gfCNCPoint2[14445] = {X -3.6095, Y 14.8821, Z -3.0000, A 0.000, B 0.000, C 0.000 }
gfCNCPoint2[14446] = {X -3.6965, Y 14.4230, Z -3.0000, A 0.000, B 0.000, C 0.000 }
gfCNCPoint2[14447] = {X -4.2194, Y 10.4573, Z -3.0000, A 0.000, B 0.000, C 0.000 }
gfCNCPoint2[14448] = {X -7.6965, Y 10.4573, Z -3.0000, A 0.000, B 0.000, C 0.000 }
gfCNCPoint2[14449] = {X -7.6965, Y 10.4573, Z 0.0000, A 0.000, B 0.000, C 0.000 }
gfCNCPoint2[14450] = {X -7.6965, Y 10.4573, Z 11.0000, A 0.000, B 0.000, C 0.000 }
gfCNCPoint2[14451] = {X -7.9918, Y 36.0072, Z 11.0000, A 0.000, B 0.000, C 0.000 }
gfCNCPoint2[14452] = {X -7.9918, Y 36.0072, Z 0.0000, A 0.000, B 0.000, C 0.000 }
gfCNCPoint2[14453] = {X -7.9918, Y 36.0072, Z -3.0000, A 0.000, B 0.000, C 0.000 }
gfCNCPoint2[14454] = {X -4.6247, Y 35.8749, Z -3.0000, A 0.000, B 0.000, C 0.000 }
gfCNCPoint2[14455] = {X -3.6965, Y 31.9841, Z -3.0000, A 0.000, B 0.000, C 0.000 }
gfCNCPoint2[14456] = {X -3.5550, Y 31.4388, Z -3.0000, A 0.000, B 0.000, C 0.000 }
gfCNCPoint2[14457] = {X -3.3921, Y 30.8996, Z -3.0000, A 0.000, B 0.000, C 0.000 }
gfCNCPoint2[14458] = {X -3.0693, Y 30.0056, Z -3.0000, A 0.000, B 0.000, C 0.000 }
gfCNCPoint2[14459] = {X -2.6877, Y 29.1351, Z -3.0000, A 0.000, B 0.000, C 0.000 }
gfCNCPoint2[14460] = {X -1.9077, Y 27.7807, Z -3.0000, A 0.000, B 0.000, C 0.000 }
gfCNCPoint2[14461] = {X -0.9348, Y 26.5574, Z -3.0000, A 0.000, B 0.000, C 0.000 }
gfCNCPoint2[14462] = {X 0.2092, Y 25.4924, Z -3.0000, A 0.000, B 0.000, C 0.000 }
gfCNCPoint2[14463] = {X 1.4989, Y 24.6096, Z -3.0000, A 0.000, B 0.000, C 0.000 }
gfCNCPoint2[14464] = {X 1.8251, Y 24.4281, Z -3.0000, A 0.000, B 0.000, C 0.000 }
gfCNCPoint2[14465] = {X 2.1575, Y 24.2584, Z -3.0000, A 0.000, B 0.000, C 0.000 }
gfCNCPoint2[14466] = {X 1.2390, Y 23.9362, Z -3.0000, A 0.000, B 0.000, C 0.000 }
gfCNCPoint2[14467] = {X 0.4229, Y 23.4056, Z -3.0000, A 0.000, B 0.000, C 0.000 }
gfCNCPoint2[14468] = {X -0.2443, Y 22.6967, Z -3.0000, A 0.000, B 0.000, C 0.000 }
gfCNCPoint2[14469] = {X -0.7246, Y 21.8500, Z -3.0000, A 0.000, B 0.000, C 0.000 }
gfCNCPoint2[14470] = {X -3.3966, Y 15.3007, Z -3.0000, A 0.000, B 0.000, C 0.000 }
gfCNCPoint2[14471] = {X -3.6235, Y 14.3620, Z -3.0000, A 0.000, B 0.000, C 0.000 }
gfCNCPoint2[14472] = {X -3.6235, Y 13.3963, Z -3.0000, A 0.000, B 0.000, C 0.000 }
gfCNCPoint2[14473] = {X -3.3966, Y 12.4576, Z -3.0000, A 0.000, B 0.000, C 0.000 }
gfCNCPoint2[14474] = {X -2.9669, Y 11.6158, Z -3.0000, A 0.000, B 0.000, C 0.000 }
gfCNCPoint2[14475] = {X -2.3551, Y 10.8955, Z -3.0000, A 0.000, B 0.000, C 0.000 }
gfCNCPoint2[14476] = {X -1.5940, Y 10.3353, Z -3.0000, A 0.000, B 0.000, C 0.000 }
gfCNCPoint2[14477] = {X -0.9968, Y 9.9946, Z -3.0000, A 0.000, B 0.000, C 0.000 }
gfCNCPoint2[14478] = {X -0.1676, Y 9.6366, Z -3.0000, A 0.000, B 0.000, C 0.000 }
gfCNCPoint2[14479] = {X 0.7200, Y 9.4699, Z -3.0000, A 0.000, B 0.000, C 0.000 }
gfCNCPoint2[14480] = {X 1.6226, Y 9.5025, Z -3.0000, A 0.000, B 0.000, C 0.000 }
gfCNCPoint2[14481] = {X 2.4959, Y 9.7329, Z -3.0000, A 0.000, B 0.000, C 0.000 }
gfCNCPoint2[14482] = {X 2.5614, Y 9.7588, Z -3.0000, A 0.000, B 0.000, C 0.000 }
gfCNCPoint2[14483] = {X 2.6265, Y 9.7860, Z -3.0000, A 0.000, B 0.000, C 0.000 }
gfCNCPoint2[14484] = {X 3.4385, Y 9.4000, Z -3.0000, A 0.000, B 0.000, C 0.000 }
gfCNCPoint2[14485] = {X 4.2752, Y 9.0711, Z -3.0000, A 0.000, B 0.000, C 0.000 }
gfCNCPoint2[14486] = {X 6.1681, Y 8.4076, Z -3.0000, A 0.000, B 0.000, C 0.000 }
gfCNCPoint2[14487] = {X 8.1112, Y 7.9101, Z -3.0000, A 0.000, B 0.000, C 0.000 }
gfCNCPoint2[14488] = {X 10.0901, Y 7.5821, Z -3.0000, A 0.000, B 0.000, C 0.000 }
gfCNCPoint2[14489] = {X 12.0898, Y 7.4262, Z -3.0000, A 0.000, B 0.000, C 0.000 }
gfCNCPoint2[14490] = {X 14.0956, Y 7.4435, Z -3.0000, A 0.000, B 0.000, C 0.000 }
gfCNCPoint2[14491] = {X 16.0924, Y 7.6340, Z -3.0000, A 0.000, B 0.000, C 0.000 }
gfCNCPoint2[14492] = {X 17.8908, Y 7.9629, Z -3.0000, A 0.000, B 0.000, C 0.000 }
gfCNCPoint2[14493] = {X 19.6442, Y 8.4808, Z -3.0000, A 0.000, B 0.000, C 0.000 }
gfCNCPoint2[14494] = {X 21.3328, Y 9.1816, Z -3.0000, A 0.000, B 0.000, C 0.000 }
gfCNCPoint2[14495] = {X 22.9375, Y 10.0576, Z -3.0000, A 0.000, B 0.000, C 0.000 }
gfCNCPoint2[14496] = {X 24.4404, Y 11.0987, Z -3.0000, A 0.000, B 0.000, C 0.000 }
gfCNCPoint2[14497] = {X 25.5052, Y 12.0298, Z -3.0000, A 0.000, B 0.000, C 0.000 }
gfCNCPoint2[14498] = {X 26.4604, Y 13.0730, Z -3.0000, A 0.000, B 0.000, C 0.000 }
gfCNCPoint2[14499] = {X 27.2942, Y 14.2157, Z -3.0000, A 0.000, B 0.000, C 0.000 }
gfCNCPoint2[14500] = {X 27.9963, Y 15.4436, Z -3.0000, A 0.000, B 0.000, C 0.000 }
gfCNCPoint2[14501] = {X 28.5581, Y 16.7417, Z -3.0000, A 0.000, B 0.000, C 0.000 }
gfCNCPoint2[14502] = {X 29.0247, Y 18.3710, Z -3.0000, A 0.000, B 0.000, C 0.000 }
gfCNCPoint2[14503] = {X 29.3015, Y 20.0431, Z -3.0000, A 0.000, B 0.000, C 0.000 }
gfCNCPoint2[14504] = {X 29.3849, Y 21.7358, Z -3.0000, A 0.000, B 0.000, C 0.000 }
gfCNCPoint2[14505] = {X 29.2739, Y 23.4270, Z -3.0000, A 0.000, B 0.000, C 0.000 }
gfCNCPoint2[14506] = {X 28.9698, Y 25.0943, Z -3.0000, A 0.000, B 0.000, C 0.000 }
gfCNCPoint2[14507] = {X 28.5023, Y 26.6013, Z -3.0000, A 0.000, B 0.000, C 0.000 }
gfCNCPoint2[14508] = {X 27.8320, Y 28.0298, Z -3.0000, A 0.000, B 0.000, C 0.000 }
gfCNCPoint2[14509] = {X 26.9717, Y 29.3525, Z -3.0000, A 0.000, B 0.000, C 0.000 }
gfCNCPoint2[14510] = {X 25.9377, Y 30.5444, Z -3.0000, A 0.000, B 0.000, C 0.000 }
gfCNCPoint2[14511] = {X 24.7496, Y 31.5828, Z -3.0000, A 0.000, B 0.000, C 0.000 }
gfCNCPoint2[14512] = {X 25.0466, Y 31.6498, Z -3.0000, A 0.000, B 0.000, C 0.000 }
gfCNCPoint2[14513] = {X 25.3378, Y 31.7388, Z -3.0000, A 0.000, B 0.000, C 0.000 }
gfCNCPoint2[14514] = {X 26.0571, Y 32.0698, Z -3.0000, A 0.000, B 0.000, C 0.000 }
gfCNCPoint2[14515] = {X 26.6990, Y 32.5334, Z -3.0000, A 0.000, B 0.000, C 0.000 }
gfCNCPoint2[14516] = {X 27.2392, Y 33.1122, Z -3.0000, A 0.000, B 0.000, C 0.000 }
gfCNCPoint2[14517] = {X 27.6575, Y 33.7845, Z -3.0000, A 0.000, B 0.000, C 0.000 }
gfCNCPoint2[14518] = {X 30.6940, Y 40.0576, Z -3.0000, A 0.000, B 0.000, C 0.000 }
gfCNCPoint2[14519] = {X 30.9967, Y 40.9162, Z -3.0000, A 0.000, B 0.000, C 0.000 }
gfCNCPoint2[14520] = {X 31.1015, Y 41.8206, Z -3.0000, A 0.000, B 0.000, C 0.000 }
gfCNCPoint2[14521] = {X 31.0032, Y 42.7257, Z -3.0000, A 0.000, B 0.000, C 0.000 }
gfCNCPoint2[14522] = {X 30.7066, Y 43.5864, Z -3.0000, A 0.000, B 0.000, C 0.000 }
gfCNCPoint2[14523] = {X 30.2265, Y 44.3600, Z -3.0000, A 0.000, B 0.000, C 0.000 }
gfCNCPoint2[14524] = {X 29.5868, Y 45.0078, Z -3.0000, A 0.000, B 0.000, C 0.000 }
gfCNCPoint2[14525] = {X 29.0507, Y 45.4413, Z -3.0000, A 0.000, B 0.000, C 0.000 }
gfCNCPoint2[14526] = {X 28.3669, Y 45.8884, Z -3.0000, A 0.000, B 0.000, C 0.000 }
gfCNCPoint2[14527] = {X 27.6079, Y 46.1908, Z -3.0000, A 0.000, B 0.000, C 0.000 }
gfCNCPoint2[14528] = {X 26.8040, Y 46.3367, Z -3.0000, A 0.000, B 0.000, C 0.000 }
gfCNCPoint2[14529] = {X 25.9872, Y 46.3201, Z -3.0000, A 0.000, B 0.000, C 0.000 }
gfCNCPoint2[14530] = {X 25.1899, Y 46.1417, Z -3.0000, A 0.000, B 0.000, C 0.000 }
gfCNCPoint2[14531] = {X 23.5977, Y 47.0009, Z -3.0000, A 0.000, B 0.000, C 0.000 }
gfCNCPoint2[14532] = {X 21.9529, Y 47.7545, Z -3.0000, A 0.000, B 0.000, C 0.000 }
gfCNCPoint2[14533] = {X 20.2625, Y 48.3992, Z -3.0000, A 0.000, B 0.000, C 0.000 }
gfCNCPoint2[14534] = {X 18.3575, Y 49.0032, Z -3.0000, A 0.000, B 0.000, C 0.000 }
gfCNCPoint2[14535] = {X 16.4065, Y 49.4364, Z -3.0000, A 0.000, B 0.000, C 0.000 }
gfCNCPoint2[14536] = {X 14.4248, Y 49.6954, Z -3.0000, A 0.000, B 0.000, C 0.000 }
gfCNCPoint2[14537] = {X 12.4280, Y 49.7781, Z -3.0000, A 0.000, B 0.000, C 0.000 }
gfCNCPoint2[14538] = {X 10.4317, Y 49.6840, Z -3.0000, A 0.000, B 0.000, C 0.000 }
gfCNCPoint2[14539] = {X 8.4515, Y 49.4137, Z -3.0000, A 0.000, B 0.000, C 0.000 }
gfCNCPoint2[14540] = {X 6.5999, Y 48.9841, Z -3.0000, A 0.000, B 0.000, C 0.000 }
gfCNCPoint2[14541] = {X 4.8081, Y 48.3494, Z -3.0000, A 0.000, B 0.000, C 0.000 }
gfCNCPoint2[14542] = {X 3.0990, Y 47.5174, Z -3.0000, A 0.000, B 0.000, C 0.000 }
gfCNCPoint2[14543] = {X 1.4941, Y 46.4988, Z -3.0000, A 0.000, B 0.000, C 0.000 }
gfCNCPoint2[14544] = {X 0.1925, Y 45.4512, Z -3.0000, A 0.000, B 0.000, C 0.000 }
gfCNCPoint2[14545] = {X -0.9646, Y 44.2459, Z -3.0000, A 0.000, B 0.000, C 0.000 }
gfCNCPoint2[14546] = {X -1.9581, Y 42.9025, Z -3.0000, A 0.000, B 0.000, C 0.000 }
gfCNCPoint2[14547] = {X -2.7718, Y 41.4432, Z -3.0000, A 0.000, B 0.000, C 0.000 }
gfCNCPoint2[14548] = {X -3.3924, Y 39.8919, Z -3.0000, A 0.000, B 0.000, C 0.000 }
gfCNCPoint2[14549] = {X -3.5562, Y 39.3526, Z -3.0000, A 0.000, B 0.000, C 0.000 }
gfCNCPoint2[14550] = {X -3.6965, Y 38.8068, Z -3.0000, A 0.000, B 0.000, C 0.000 }
gfCNCPoint2[14551] = {X -4.6086, Y 34.9122, Z -3.0000, A 0.000, B 0.000, C 0.000 }
gfCNCPoint2[14552] = {X -7.9997, Y 34.8247, Z -3.0000, A 0.000, B 0.000, C 0.000 }
gfCNCPoint2[14553] = {X -7.9997, Y 34.8247, Z 0.0000, A 0.000, B 0.000, C 0.000 }
gfCNCPoint2[14554] = {X -7.9997, Y 34.8247, Z 11.0000, A 0.000, B 0.000, C 0.000 }
gfCNCPoint2[14555] = {X -7.9666, Y 36.4869, Z 11.0000, A 0.000, B 0.000, C 0.000 }
gfCNCPoint2[14556] = {X -7.9666, Y 36.4869, Z 0.0000, A 0.000, B 0.000, C 0.000 }
gfCNCPoint2[14557] = {X -7.9666, Y 36.4869, Z -3.0000, A 0.000, B 0.000, C 0.000 }
gfCNCPoint2[14558] = {X -4.5273, Y 36.2607, Z -3.0000, A 0.000, B 0.000, C 0.000 }
gfCNCPoint2[14559] = {X -3.6965, Y 32.3479, Z -3.0000, A 0.000, B 0.000, C 0.000 }
gfCNCPoint2[14560] = {X -3.5247, Y 31.6311, Z -3.0000, A 0.000, B 0.000, C 0.000 }
gfCNCPoint2[14561] = {X -3.3160, Y 30.9243, Z -3.0000, A 0.000, B 0.000, C 0.000 }
gfCNCPoint2[14562] = {X -2.9950, Y 30.0353, Z -3.0000, A 0.000, B 0.000, C 0.000 }
gfCNCPoint2[14563] = {X -2.6155, Y 29.1697, Z -3.0000, A 0.000, B 0.000, C 0.000 }
gfCNCPoint2[14564] = {X -1.8415, Y 27.8256, Z -3.0000, A 0.000, B 0.000, C 0.000 }
gfCNCPoint2[14565] = {X -0.8761, Y 26.6117, Z -3.0000, A 0.000, B 0.000, C 0.000 }
gfCNCPoint2[14566] = {X 0.2592, Y 25.5549, Z -3.0000, A 0.000, B 0.000, C 0.000 }
gfCNCPoint2[14567] = {X 1.5391, Y 24.6788, Z -3.0000, A 0.000, B 0.000, C 0.000 }
gfCNCPoint2[14568] = {X 1.9710, Y 24.4418, Z -3.0000, A 0.000, B 0.000, C 0.000 }
gfCNCPoint2[14569] = {X 2.4136, Y 24.2255, Z -3.0000, A 0.000, B 0.000, C 0.000 }
gfCNCPoint2[14570] = {X 1.6216, Y 24.0151, Z -3.0000, A 0.000, B 0.000, C 0.000 }
gfCNCPoint2[14571] = {X 0.8890, Y 23.6478, Z -3.0000, A 0.000, B 0.000, C 0.000 }
gfCNCPoint2[14572] = {X 0.2467, Y 23.1388, Z -3.0000, A 0.000, B 0.000, C 0.000 }
gfCNCPoint2[14573] = {X -0.2784, Y 22.5096, Z -3.0000, A 0.000, B 0.000, C 0.000 }
gfCNCPoint2[14574] = {X -0.6642, Y 21.7866, Z -3.0000, A 0.000, B 0.000, C 0.000 }
gfCNCPoint2[14575] = {X -3.2754, Y 15.3911, Z -3.0000, A 0.000, B 0.000, C 0.000 }
gfCNCPoint2[14576] = {X -3.2990, Y 15.3321, Z -3.0000, A 0.000, B 0.000, C 0.000 }
gfCNCPoint2[14577] = {X -3.3216, Y 15.2728, Z -3.0000, A 0.000, B 0.000, C 0.000 }
gfCNCPoint2[14578] = {X -3.5441, Y 14.3525, Z -3.0000, A 0.000, B 0.000, C 0.000 }
gfCNCPoint2[14579] = {X -3.5441, Y 13.4057, Z -3.0000, A 0.000, B 0.000, C 0.000 }
gfCNCPoint2[14580] = {X -3.3216, Y 12.4855, Z -3.0000, A 0.000, B 0.000, C 0.000 }
gfCNCPoint2[14581] = {X -2.9003, Y 11.6602, Z -3.0000, A 0.000, B 0.000, C 0.000 }
gfCNCPoint2[14582] = {X -2.3006, Y 10.9540, Z -3.0000, A 0.000, B 0.000, C 0.000 }
gfCNCPoint2[14583] = {X -1.5544, Y 10.4048, Z -3.0000, A 0.000, B 0.000, C 0.000 }
gfCNCPoint2[14584] = {X -0.9063, Y 10.0355, Z -3.0000, A 0.000, B 0.000, C 0.000 }
gfCNCPoint2[14585] = {X -0.1023, Y 9.7006, Z -3.0000, A 0.000, B 0.000, C 0.000 }
gfCNCPoint2[14586] = {X 0.7551, Y 9.5476, Z -3.0000, A 0.000, B 0.000, C 0.000 }
gfCNCPoint2[14587] = {X 1.6253, Y 9.5838, Z -3.0000, A 0.000, B 0.000, C 0.000 }
gfCNCPoint2[14588] = {X 2.4670, Y 9.8075, Z -3.0000, A 0.000, B 0.000, C 0.000 }
gfCNCPoint2[14589] = {X 2.5487, Y 9.8401, Z -3.0000, A 0.000, B 0.000, C 0.000 }
gfCNCPoint2[14590] = {X 2.6297, Y 9.8745, Z -3.0000, A 0.000, B 0.000, C 0.000 }
gfCNCPoint2[14591] = {X 3.4566, Y 9.4794, Z -3.0000, A 0.000, B 0.000, C 0.000 }
gfCNCPoint2[14592] = {X 4.3093, Y 9.1438, Z -3.0000, A 0.000, B 0.000, C 0.000 }
gfCNCPoint2[14593] = {X 6.1951, Y 8.4832, Z -3.0000, A 0.000, B 0.000, C 0.000 }
gfCNCPoint2[14594] = {X 8.1309, Y 7.9878, Z -3.0000, A 0.000, B 0.000, C 0.000 }
gfCNCPoint2[14595] = {X 10.1022, Y 7.6613, Z -3.0000, A 0.000, B 0.000, C 0.000 }
gfCNCPoint2[14596] = {X 12.0944, Y 7.5062, Z -3.0000, A 0.000, B 0.000, C 0.000 }
gfCNCPoint2[14597] = {X 14.0924, Y 7.5235, Z -3.0000, A 0.000, B 0.000, C 0.000 }
gfCNCPoint2[14598] = {X 16.0816, Y 7.7132, Z -3.0000, A 0.000, B 0.000, C 0.000 }
gfCNCPoint2[14599] = {X 16.4812, Y 7.7686, Z -3.0000, A 0.000, B 0.000, C 0.000 }
gfCNCPoint2[14600] = {X 18.1851, Y 8.1178, Z -3.0000, A 0.000, B 0.000, C 0.000 }
gfCNCPoint2[14601] = {X 19.8449, Y 8.6380, Z -3.0000, A 0.000, B 0.000, C 0.000 }
gfCNCPoint2[14602] = {X 21.4433, Y 9.3237, Z -3.0000, A 0.000, B 0.000, C 0.000 }
gfCNCPoint2[14603] = {X 22.9641, Y 10.1679, Z -3.0000, A 0.000, B 0.000, C 0.000 }
gfCNCPoint2[14604] = {X 24.3914, Y 11.1620, Z -3.0000, A 0.000, B 0.000, C 0.000 }
gfCNCPoint2[14605] = {X 25.4494, Y 12.0871, Z -3.0000, A 0.000, B 0.000, C 0.000 }
gfCNCPoint2[14606] = {X 26.3985, Y 13.1236, Z -3.0000, A 0.000, B 0.000, C 0.000 }
gfCNCPoint2[14607] = {X 27.2269, Y 14.2589, Z -3.0000, A 0.000, B 0.000, C 0.000 }
gfCNCPoint2[14608] = {X 27.9245, Y 15.4790, Z -3.0000, A 0.000, B 0.000, C 0.000 }
gfCNCPoint2[14609] = {X 28.4828, Y 16.7687, Z -3.0000, A 0.000, B 0.000, C 0.000 }
gfCNCPoint2[14610] = {X 28.9468, Y 18.3894, Z -3.0000, A 0.000, B 0.000, C 0.000 }
gfCNCPoint2[14611] = {X 29.2220, Y 20.0524, Z -3.0000, A 0.000, B 0.000, C 0.000 }
gfCNCPoint2[14612] = {X 29.3049, Y 21.7361, Z -3.0000, A 0.000, B 0.000, C 0.000 }
gfCNCPoint2[14613] = {X 29.1943, Y 23.4182, Z -3.0000, A 0.000, B 0.000, C 0.000 }
gfCNCPoint2[14614] = {X 28.8918, Y 25.0766, Z -3.0000, A 0.000, B 0.000, C 0.000 }
gfCNCPoint2[14615] = {X 28.4139, Y 26.6079, Z -3.0000, A 0.000, B 0.000, C 0.000 }
gfCNCPoint2[14616] = {X 27.7252, Y 28.0568, Z -3.0000, A 0.000, B 0.000, C 0.000 }
gfCNCPoint2[14617] = {X 26.8394, Y 29.3943, Z -3.0000, A 0.000, B 0.000, C 0.000 }
gfCNCPoint2[14618] = {X 25.7741, Y 30.5938, Z -3.0000, A 0.000, B 0.000, C 0.000 }
gfCNCPoint2[14619] = {X 24.5506, Y 31.6314, Z -3.0000, A 0.000, B 0.000, C 0.000 }
gfCNCPoint2[14620] = {X 24.9356, Y 31.7043, Z -3.0000, A 0.000, B 0.000, C 0.000 }
gfCNCPoint2[14621] = {X 25.3116, Y 31.8144, Z -3.0000, A 0.000, B 0.000, C 0.000 }
gfCNCPoint2[14622] = {X 26.0242, Y 32.1432, Z -3.0000, A 0.000, B 0.000, C 0.000 }
gfCNCPoint2[14623] = {X 26.6589, Y 32.6047, Z -3.0000, A 0.000, B 0.000, C 0.000 }
gfCNCPoint2[14624] = {X 27.1913, Y 33.1814, Z -3.0000, A 0.000, B 0.000, C 0.000 }
gfCNCPoint2[14625] = {X 27.6008, Y 33.8508, Z -3.0000, A 0.000, B 0.000, C 0.000 }
gfCNCPoint2[14626] = {X 30.6220, Y 40.0925, Z -3.0000, A 0.000, B 0.000, C 0.000 }
gfCNCPoint2[14627] = {X 30.9188, Y 40.9342, Z -3.0000, A 0.000, B 0.000, C 0.000 }
gfCNCPoint2[14628] = {X 31.0215, Y 41.8209, Z -3.0000, A 0.000, B 0.000, C 0.000 }
gfCNCPoint2[14629] = {X 30.9251, Y 42.7082, Z -3.0000, A 0.000, B 0.000, C 0.000 }
gfCNCPoint2[14630] = {X 30.6343, Y 43.5521, Z -3.0000, A 0.000, B 0.000, C 0.000 }
gfCNCPoint2[14631] = {X 30.1637, Y 44.3105, Z -3.0000, A 0.000, B 0.000, C 0.000 }
gfCNCPoint2[14632] = {X 29.5365, Y 44.9456, Z -3.0000, A 0.000, B 0.000, C 0.000 }
gfCNCPoint2[14633] = {X 29.0005, Y 45.3790, Z -3.0000, A 0.000, B 0.000, C 0.000 }
gfCNCPoint2[14634] = {X 28.1799, Y 45.8914, Z -3.0000, A 0.000, B 0.000, C 0.000 }
gfCNCPoint2[14635] = {X 27.2606, Y 46.1927, Z -3.0000, A 0.000, B 0.000, C 0.000 }
gfCNCPoint2[14636] = {X 26.2959, Y 46.2655, Z -3.0000, A 0.000, B 0.000, C 0.000 }
gfCNCPoint2[14637] = {X 25.3418, Y 46.1055, Z -3.0000, A 0.000, B 0.000, C 0.000 }
gfCNCPoint2[14638] = {X 25.2611, Y 46.0807, Z -3.0000, A 0.000, B 0.000, C 0.000 }
gfCNCPoint2[14639] = {X 25.1810, Y 46.0543, Z -3.0000, A 0.000, B 0.000, C 0.000 }
gfCNCPoint2[14640] = {X 23.5837, Y 46.9185, Z -3.0000, A 0.000, B 0.000, C 0.000 }
gfCNCPoint2[14641] = {X 21.9332, Y 47.6760, Z -3.0000, A 0.000, B 0.000, C 0.000 }
gfCNCPoint2[14642] = {X 20.2365, Y 48.3236, Z -3.0000, A 0.000, B 0.000, C 0.000 }
gfCNCPoint2[14643] = {X 19.5440, Y 48.5625, Z -3.0000, A 0.000, B 0.000, C 0.000 }
gfCNCPoint2[14644] = {X 17.3812, Y 49.1590, Z -3.0000, A 0.000, B 0.000, C 0.000 }
gfCNCPoint2[14645] = {X 15.1697, Y 49.5371, Z -3.0000, A 0.000, B 0.000, C 0.000 }
gfCNCPoint2[14646] = {X 12.9315, Y 49.6931, Z -3.0000, A 0.000, B 0.000, C 0.000 }
gfCNCPoint2[14647] = {X 10.6889, Y 49.6254, Z -3.0000, A 0.000, B 0.000, C 0.000 }
gfCNCPoint2[14648] = {X 8.4642, Y 49.3347, Z -3.0000, A 0.000, B 0.000, C 0.000 }
gfCNCPoint2[14649] = {X 6.6212, Y 48.9070, Z -3.0000, A 0.000, B 0.000, C 0.000 }
gfCNCPoint2[14650] = {X 4.8378, Y 48.2751, Z -3.0000, A 0.000, B 0.000, C 0.000 }
gfCNCPoint2[14651] = {X 3.1367, Y 47.4469, Z -3.0000, A 0.000, B 0.000, C 0.000 }
gfCNCPoint2[14652] = {X 1.5394, Y 46.4329, Z -3.0000, A 0.000, B 0.000, C 0.000 }
gfCNCPoint2[14653] = {X 0.2460, Y 45.3917, Z -3.0000, A 0.000, B 0.000, C 0.000 }
gfCNCPoint2[14654] = {X -0.9038, Y 44.1938, Z -3.0000, A 0.000, B 0.000, C 0.000 }
gfCNCPoint2[14655] = {X -1.8911, Y 42.8588, Z -3.0000, A 0.000, B 0.000, C 0.000 }
gfCNCPoint2[14656] = {X -2.6997, Y 41.4086, Z -3.0000, A 0.000, B 0.000, C 0.000 }
gfCNCPoint2[14657] = {X -3.3164, Y 39.8670, Z -3.0000, A 0.000, B 0.000, C 0.000 }
gfCNCPoint2[14658] = {X -3.5270, Y 39.1557, Z -3.0000, A 0.000, B 0.000, C 0.000 }
gfCNCPoint2[14659] = {X -3.6965, Y 38.4336, Z -3.0000, A 0.000, B 0.000, C 0.000 }
gfCNCPoint2[14660] = {X -4.4992, Y 34.5150, Z -3.0000, A 0.000, B 0.000, C 0.000 }
gfCNCPoint2[14661] = {X -7.9803, Y 34.3303, Z -3.0000, A 0.000, B 0.000, C 0.000 }
gfCNCPoint2[14662] = {X -7.9803, Y 34.3303, Z 0.0000, A 0.000, B 0.000, C 0.000 }
gfCNCPoint2[14663] = {X -7.9803, Y 34.3303, Z 11.0000, A 0.000, B 0.000, C 0.000 }
gfCNCPoint2[14664] = {X 39.8138, Y 26.4139, Z 11.0000, A 0.000, B 0.000, C 0.000 }
gfCNCPoint2[14665] = {X 39.8138, Y 26.4139, Z 0.0000, A 0.000, B 0.000, C 0.000 }
gfCNCPoint2[14666] = {X 39.8138, Y 26.4139, Z -3.0000, A 0.000, B 0.000, C 0.000 }
gfCNCPoint2[14667] = {X 43.6372, Y 27.8379, Z -3.0000, A 0.000, B 0.000, C 0.000 }
gfCNCPoint2[14668] = {X 48.2902, Y 15.3446, Z -3.0000, A 0.000, B 0.000, C 0.000 }
gfCNCPoint2[14669] = {X 47.9079, Y 14.6186, Z -3.0000, A 0.000, B 0.000, C 0.000 }
gfCNCPoint2[14670] = {X 47.6697, Y 13.8334, Z -3.0000, A 0.000, B 0.000, C 0.000 }
gfCNCPoint2[14671] = {X 47.5844, Y 13.0173, Z -3.0000, A 0.000, B 0.000, C 0.000 }
gfCNCPoint2[14672] = {X 47.5842, Y 12.1868, Z -3.0000, A 0.000, B 0.000, C 0.000 }
gfCNCPoint2[14673] = {X 47.6925, Y 11.2255, Z -3.0000, A 0.000, B 0.000, C 0.000 }
gfCNCPoint2[14674] = {X 48.0120, Y 10.3125, Z -3.0000, A 0.000, B 0.000, C 0.000 }
gfCNCPoint2[14675] = {X 48.5267, Y 9.4933, Z -3.0000, A 0.000, B 0.000, C 0.000 }
gfCNCPoint2[14676] = {X 49.2107, Y 8.8093, Z -3.0000, A 0.000, B 0.000, C 0.000 }
gfCNCPoint2[14677] = {X 50.0298, Y 8.2946, Z -3.0000, A 0.000, B 0.000, C 0.000 }
gfCNCPoint2[14678] = {X 50.9429, Y 7.9751, Z -3.0000, A 0.000, B 0.000, C 0.000 }
gfCNCPoint2[14679] = {X 51.9042, Y 7.8668, Z -3.0000, A 0.000, B 0.000, C 0.000 }
gfCNCPoint2[14680] = {X 59.6221, Y 7.8668, Z -3.0000, A 0.000, B 0.000, C 0.000 }
gfCNCPoint2[14681] = {X 60.5834, Y 7.9751, Z -3.0000, A 0.000, B 0.000, C 0.000 }
gfCNCPoint2[14682] = {X 61.4965, Y 8.2946, Z -3.0000, A 0.000, B 0.000, C 0.000 }
gfCNCPoint2[14683] = {X 62.3156, Y 8.8093, Z -3.0000, A 0.000, B 0.000, C 0.000 }
gfCNCPoint2[14684] = {X 62.9996, Y 9.4933, Z -3.0000, A 0.000, B 0.000, C 0.000 }
gfCNCPoint2[14685] = {X 63.5143, Y 10.3124, Z -3.0000, A 0.000, B 0.000, C 0.000 }
gfCNCPoint2[14686] = {X 63.8338, Y 11.2255, Z -3.0000, A 0.000, B 0.000, C 0.000 }
gfCNCPoint2[14687] = {X 63.9421, Y 12.1868, Z -3.0000, A 0.000, B 0.000, C 0.000 }
gfCNCPoint2[14688] = {X 63.9421, Y 12.9781, Z -3.0000, A 0.000, B 0.000, C 0.000 }
gfCNCPoint2[14689] = {X 63.8583, Y 13.8249, Z -3.0000, A 0.000, B 0.000, C 0.000 }
gfCNCPoint2[14690] = {X 63.6101, Y 14.6388, Z -3.0000, A 0.000, B 0.000, C 0.000 }
gfCNCPoint2[14691] = {X 63.2072, Y 15.3883, Z -3.0000, A 0.000, B 0.000, C 0.000 }
gfCNCPoint2[14692] = {X 63.4251, Y 15.9633, Z -3.0000, A 0.000, B 0.000, C 0.000 }
gfCNCPoint2[14693] = {X 66.0345, Y 22.8874, Z -3.0000, A 0.000, B 0.000, C 0.000 }
gfCNCPoint2[14694] = {X 72.2090, Y 39.5004, Z -3.0000, A 0.000, B 0.000, C 0.000 }
gfCNCPoint2[14695] = {X 72.5142, Y 40.2679, Z -3.0000, A 0.000, B 0.000, C 0.000 }
gfCNCPoint2[14696] = {X 73.3588, Y 40.7697, Z -3.0000, A 0.000, B 0.000, C 0.000 }
gfCNCPoint2[14697] = {X 74.0682, Y 41.4493, Z -3.0000, A 0.000, B 0.000, C 0.000 }
gfCNCPoint2[14698] = {X 74.6058, Y 42.2716, Z -3.0000, A 0.000, B 0.000, C 0.000 }
gfCNCPoint2[14699] = {X 74.9436, Y 43.1942, Z -3.0000, A 0.000, B 0.000, C 0.000 }
gfCNCPoint2[14700] = {X 75.0643, Y 44.1692, Z -3.0000, A 0.000, B 0.000, C 0.000 }
gfCNCPoint2[14701] = {X 75.0645, Y 45.0000, Z -3.0000, A 0.000, B 0.000, C 0.000 }
gfCNCPoint2[14702] = {X 74.9561, Y 45.9613, Z -3.0000, A 0.000, B 0.000, C 0.000 }
gfCNCPoint2[14703] = {X 74.6366, Y 46.8744, Z -3.0000, A 0.000, B 0.000, C 0.000 }
gfCNCPoint2[14704] = {X 74.1220, Y 47.6935, Z -3.0000, A 0.000, B 0.000, C 0.000 }
gfCNCPoint2[14705] = {X 73.4379, Y 48.3775, Z -3.0000, A 0.000, B 0.000, C 0.000 }
gfCNCPoint2[14706] = {X 72.6188, Y 48.8922, Z -3.0000, A 0.000, B 0.000, C 0.000 }
gfCNCPoint2[14707] = {X 71.7057, Y 49.2117, Z -3.0000, A 0.000, B 0.000, C 0.000 }
gfCNCPoint2[14708] = {X 70.7445, Y 49.3200, Z -3.0000, A 0.000, B 0.000, C 0.000 }
gfCNCPoint2[14709] = {X 64.1851, Y 49.3200, Z -3.0000, A 0.000, B 0.000, C 0.000 }
gfCNCPoint2[14710] = {X 63.2238, Y 49.2117, Z -3.0000, A 0.000, B 0.000, C 0.000 }
gfCNCPoint2[14711] = {X 62.3108, Y 48.8922, Z -3.0000, A 0.000, B 0.000, C 0.000 }
gfCNCPoint2[14712] = {X 61.4917, Y 48.3775, Z -3.0000, A 0.000, B 0.000, C 0.000 }
gfCNCPoint2[14713] = {X 60.8076, Y 47.6935, Z -3.0000, A 0.000, B 0.000, C 0.000 }
gfCNCPoint2[14714] = {X 60.2929, Y 46.8744, Z -3.0000, A 0.000, B 0.000, C 0.000 }
gfCNCPoint2[14715] = {X 59.9734, Y 45.9613, Z -3.0000, A 0.000, B 0.000, C 0.000 }
gfCNCPoint2[14716] = {X 59.8651, Y 45.0000, Z -3.0000, A 0.000, B 0.000, C 0.000 }
gfCNCPoint2[14717] = {X 59.8651, Y 44.2084, Z -3.0000, A 0.000, B 0.000, C 0.000 }
gfCNCPoint2[14718] = {X 59.9520, Y 43.3500, Z -3.0000, A 0.000, B 0.000, C 0.000 }
gfCNCPoint2[14719] = {X 60.2077, Y 42.5259, Z -3.0000, A 0.000, B 0.000, C 0.000 }
gfCNCPoint2[14720] = {X 60.6221, Y 41.7691, Z -3.0000, A 0.000, B 0.000, C 0.000 }
gfCNCPoint2[14721] = {X 60.0072, Y 40.0892, Z -3.0000, A 0.000, B 0.000, C 0.000 }
gfCNCPoint2[14722] = {X 52.0767, Y 40.0892, Z -3.0000, A 0.000, B 0.000, C 0.000 }
gfCNCPoint2[14723] = {X 51.3341, Y 42.0842, Z -3.0000, A 0.000, B 0.000, C 0.000 }
gfCNCPoint2[14724] = {X 51.3373, Y 42.0894, Z -3.0000, A 0.000, B 0.000, C 0.000 }
gfCNCPoint2[14725] = {X 51.6388, Y 42.7490, Z -3.0000, A 0.000, B 0.000, C 0.000 }
gfCNCPoint2[14726] = {X 51.8257, Y 43.4498, Z -3.0000, A 0.000, B 0.000, C 0.000 }
gfCNCPoint2[14727] = {X 51.8928, Y 44.1720, Z -3.0000, A 0.000, B 0.000, C 0.000 }
gfCNCPoint2[14728] = {X 51.8929, Y 45.0000, Z -3.0000, A 0.000, B 0.000, C 0.000 }
gfCNCPoint2[14729] = {X 51.7846, Y 45.9613, Z -3.0000, A 0.000, B 0.000, C 0.000 }
gfCNCPoint2[14730] = {X 51.4651, Y 46.8744, Z -3.0000, A 0.000, B 0.000, C 0.000 }
gfCNCPoint2[14731] = {X 50.9504, Y 47.6935, Z -3.0000, A 0.000, B 0.000, C 0.000 }
gfCNCPoint2[14732] = {X 50.2664, Y 48.3775, Z -3.0000, A 0.000, B 0.000, C 0.000 }
gfCNCPoint2[14733] = {X 49.4473, Y 48.8922, Z -3.0000, A 0.000, B 0.000, C 0.000 }
gfCNCPoint2[14734] = {X 48.5342, Y 49.2117, Z -3.0000, A 0.000, B 0.000, C 0.000 }
gfCNCPoint2[14735] = {X 47.5729, Y 49.3200, Z -3.0000, A 0.000, B 0.000, C 0.000 }
gfCNCPoint2[14736] = {X 40.6393, Y 49.3200, Z -3.0000, A 0.000, B 0.000, C 0.000 }
gfCNCPoint2[14737] = {X 39.6780, Y 49.2117, Z -3.0000, A 0.000, B 0.000, C 0.000 }
gfCNCPoint2[14738] = {X 38.7649, Y 48.8922, Z -3.0000, A 0.000, B 0.000, C 0.000 }
gfCNCPoint2[14739] = {X 37.9458, Y 48.3775, Z -3.0000, A 0.000, B 0.000, C 0.000 }
gfCNCPoint2[14740] = {X 37.2618, Y 47.6935, Z -3.0000, A 0.000, B 0.000, C 0.000 }
gfCNCPoint2[14741] = {X 36.7471, Y 46.8744, Z -3.0000, A 0.000, B 0.000, C 0.000 }
gfCNCPoint2[14742] = {X 36.4276, Y 45.9613, Z -3.0000, A 0.000, B 0.000, C 0.000 }
gfCNCPoint2[14743] = {X 36.3193, Y 45.0000, Z -3.0000, A 0.000, B 0.000, C 0.000 }
gfCNCPoint2[14744] = {X 36.3193, Y 44.2086, Z -3.0000, A 0.000, B 0.000, C 0.000 }
gfCNCPoint2[14745] = {X 36.4325, Y 43.2262, Z -3.0000, A 0.000, B 0.000, C 0.000 }
gfCNCPoint2[14746] = {X 36.7662, Y 42.2952, Z -3.0000, A 0.000, B 0.000, C 0.000 }
gfCNCPoint2[14747] = {X 37.3029, Y 41.4646, Z -3.0000, A 0.000, B 0.000, C 0.000 }
gfCNCPoint2[14748] = {X 38.0144, Y 40.7777, Z -3.0000, A 0.000, B 0.000, C 0.000 }
gfCNCPoint2[14749] = {X 38.8635, Y 40.2707, Z -3.0000, A 0.000, B 0.000, C 0.000 }
gfCNCPoint2[14750] = {X 38.9643, Y 40.1703, Z -3.0000, A 0.000, B 0.000, C 0.000 }
gfCNCPoint2[14751] = {X 39.5382, Y 38.8092, Z -3.0000, A 0.000, B 0.000, C 0.000 }
gfCNCPoint2[14752] = {X 40.0650, Y 37.4293, Z -3.0000, A 0.000, B 0.000, C 0.000 }
gfCNCPoint2[14753] = {X 43.6372, Y 27.8379, Z -3.0000, A 0.000, B 0.000, C 0.000 }
gfCNCPoint2[14754] = {X 39.8887, Y 26.4418, Z -3.0000, A 0.000, B 0.000, C 0.000 }
gfCNCPoint2[14755] = {X 43.7122, Y 27.8658, Z -3.0000, A 0.000, B 0.000, C 0.000 }
gfCNCPoint2[14756] = {X 48.3793, Y 15.3344, Z -3.0000, A 0.000, B 0.000, C 0.000 }
gfCNCPoint2[14757] = {X 47.9922, Y 14.6130, Z -3.0000, A 0.000, B 0.000, C 0.000 }
gfCNCPoint2[14758] = {X 47.7508, Y 13.8307, Z -3.0000, A 0.000, B 0.000, C 0.000 }
gfCNCPoint2[14759] = {X 47.6644, Y 13.0166, Z -3.0000, A 0.000, B 0.000, C 0.000 }
gfCNCPoint2[14760] = {X 47.6642, Y 12.1868, Z -3.0000, A 0.000, B 0.000, C 0.000 }
gfCNCPoint2[14761] = {X 47.7705, Y 11.2433, Z -3.0000, A 0.000, B 0.000, C 0.000 }
gfCNCPoint2[14762] = {X 48.0841, Y 10.3472, Z -3.0000, A 0.000, B 0.000, C 0.000 }
gfCNCPoint2[14763] = {X 48.5893, Y 9.5432, Z -3.0000, A 0.000, B 0.000, C 0.000 }
gfCNCPoint2[14764] = {X 49.2606, Y 8.8719, Z -3.0000, A 0.000, B 0.000, C 0.000 }
gfCNCPoint2[14765] = {X 50.0646, Y 8.3667, Z -3.0000, A 0.000, B 0.000, C 0.000 }
gfCNCPoint2[14766] = {X 50.9607, Y 8.0531, Z -3.0000, A 0.000, B 0.000, C 0.000 }
gfCNCPoint2[14767] = {X 51.9042, Y 7.9468, Z -3.0000, A 0.000, B 0.000, C 0.000 }
gfCNCPoint2[14768] = {X 59.6221, Y 7.9468, Z -3.0000, A 0.000, B 0.000, C 0.000 }
gfCNCPoint2[14769] = {X 60.5656, Y 8.0531, Z -3.0000, A 0.000, B 0.000, C 0.000 }
gfCNCPoint2[14770] = {X 61.4618, Y 8.3667, Z -3.0000, A 0.000, B 0.000, C 0.000 }
gfCNCPoint2[14771] = {X 62.2657, Y 8.8718, Z -3.0000, A 0.000, B 0.000, C 0.000 }
gfCNCPoint2[14772] = {X 62.9371, Y 9.5432, Z -3.0000, A 0.000, B 0.000, C 0.000 }
gfCNCPoint2[14773] = {X 63.4422, Y 10.3471, Z -3.0000, A 0.000, B 0.000, C 0.000 }
gfCNCPoint2[14774] = {X 63.7558, Y 11.2433, Z -3.0000, A 0.000, B 0.000, C 0.000 }
gfCNCPoint2[14775] = {X 63.8621, Y 12.1868, Z -3.0000, A 0.000, B 0.000, C 0.000 }
gfCNCPoint2[14776] = {X 63.8621, Y 12.9781, Z -3.0000, A 0.000, B 0.000, C 0.000 }
gfCNCPoint2[14777] = {X 63.7771, Y 13.8227, Z -3.0000, A 0.000, B 0.000, C 0.000 }
gfCNCPoint2[14778] = {X 63.5256, Y 14.6334, Z -3.0000, A 0.000, B 0.000, C 0.000 }
gfCNCPoint2[14779] = {X 63.1177, Y 15.3777, Z -3.0000, A 0.000, B 0.000, C 0.000 }
gfCNCPoint2[14780] = {X 63.3503, Y 15.9916, Z -3.0000, A 0.000, B 0.000, C 0.000 }
gfCNCPoint2[14781] = {X 65.9595, Y 22.9155, Z -3.0000, A 0.000, B 0.000, C 0.000 }
gfCNCPoint2[14782] = {X 72.1343, Y 39.5291, Z -3.0000, A 0.000, B 0.000, C 0.000 }
gfCNCPoint2[14783] = {X 72.4519, Y 40.3278, Z -3.0000, A 0.000, B 0.000, C 0.000 }
gfCNCPoint2[14784] = {X 73.2898, Y 40.8178, Z -3.0000, A 0.000, B 0.000, C 0.000 }
gfCNCPoint2[14785] = {X 73.9943, Y 41.4855, Z -3.0000, A 0.000, B 0.000, C 0.000 }
gfCNCPoint2[14786] = {X 74.5285, Y 42.2960, Z -3.0000, A 0.000, B 0.000, C 0.000 }
gfCNCPoint2[14787] = {X 74.8643, Y 43.2067, Z -3.0000, A 0.000, B 0.000, C 0.000 }
gfCNCPoint2[14788] = {X 74.9843, Y 44.1699, Z -3.0000, A 0.000, B 0.000, C 0.000 }
gfCNCPoint2[14789] = {X 74.9845, Y 45.0000, Z -3.0000, A 0.000, B 0.000, C 0.000 }
gfCNCPoint2[14790] = {X 74.8782, Y 45.9435, Z -3.0000, A 0.000, B 0.000, C 0.000 }
gfCNCPoint2[14791] = {X 74.5646, Y 46.8397, Z -3.0000, A 0.000, B 0.000, C 0.000 }
gfCNCPoint2[14792] = {X 74.0594, Y 47.6436, Z -3.0000, A 0.000, B 0.000, C 0.000 }
gfCNCPoint2[14793] = {X 73.3881, Y 48.3150, Z -3.0000, A 0.000, B 0.000, C 0.000 }
gfCNCPoint2[14794] = {X 72.5841, Y 48.8201, Z -3.0000, A 0.000, B 0.000, C 0.000 }
gfCNCPoint2[14795] = {X 71.6879, Y 49.1337, Z -3.0000, A 0.000, B 0.000, C 0.000 }
gfCNCPoint2[14796] = {X 70.7445, Y 49.2400, Z -3.0000, A 0.000, B 0.000, C 0.000 }
gfCNCPoint2[14797] = {X 64.1851, Y 49.2400, Z -3.0000, A 0.000, B 0.000, C 0.000 }
gfCNCPoint2[14798] = {X 63.2416, Y 49.1337, Z -3.0000, A 0.000, B 0.000, C 0.000 }
gfCNCPoint2[14799] = {X 62.3455, Y 48.8201, Z -3.0000, A 0.000, B 0.000, C 0.000 }
gfCNCPoint2[14800] = {X 61.5415, Y 48.3150, Z -3.0000, A 0.000, B 0.000, C 0.000 }
gfCNCPoint2[14801] = {X 60.8702, Y 47.6436, Z -3.0000, A 0.000, B 0.000, C 0.000 }
gfCNCPoint2[14802] = {X 60.3650, Y 46.8397, Z -3.0000, A 0.000, B 0.000, C 0.000 }
gfCNCPoint2[14803] = {X 60.0514, Y 45.9435, Z -3.0000, A 0.000, B 0.000, C 0.000 }
gfCNCPoint2[14804] = {X 59.9451, Y 45.0000, Z -3.0000, A 0.000, B 0.000, C 0.000 }
gfCNCPoint2[14805] = {X 59.9451, Y 44.2085, Z -3.0000, A 0.000, B 0.000, C 0.000 }
gfCNCPoint2[14806] = {X 60.0332, Y 43.3525, Z -3.0000, A 0.000, B 0.000, C 0.000 }
gfCNCPoint2[14807] = {X 60.2922, Y 42.5320, Z -3.0000, A 0.000, B 0.000, C 0.000 }
gfCNCPoint2[14808] = {X 60.7115, Y 41.7806, Z -3.0000, A 0.000, B 0.000, C 0.000 }
gfCNCPoint2[14809] = {X 60.0631, Y 40.0092, Z -3.0000, A 0.000, B 0.000, C 0.000 }
gfCNCPoint2[14810] = {X 52.0212, Y 40.0092, Z -3.0000, A 0.000, B 0.000, C 0.000 }
gfCNCPoint2[14811] = {X 51.2457, Y 42.0925, Z -3.0000, A 0.000, B 0.000, C 0.000 }
gfCNCPoint2[14812] = {X 51.2682, Y 42.1297, Z -3.0000, A 0.000, B 0.000, C 0.000 }
gfCNCPoint2[14813] = {X 51.5638, Y 42.7768, Z -3.0000, A 0.000, B 0.000, C 0.000 }
gfCNCPoint2[14814] = {X 51.7470, Y 43.4643, Z -3.0000, A 0.000, B 0.000, C 0.000 }
gfCNCPoint2[14815] = {X 51.8128, Y 44.1726, Z -3.0000, A 0.000, B 0.000, C 0.000 }
gfCNCPoint2[14816] = {X 51.8129, Y 45.0000, Z -3.0000, A 0.000, B 0.000, C 0.000 }
gfCNCPoint2[14817] = {X 51.7066, Y 45.9435, Z -3.0000, A 0.000, B 0.000, C 0.000 }
gfCNCPoint2[14818] = {X 51.3930, Y 46.8397, Z -3.0000, A 0.000, B 0.000, C 0.000 }
gfCNCPoint2[14819] = {X 50.8879, Y 47.6436, Z -3.0000, A 0.000, B 0.000, C 0.000 }
gfCNCPoint2[14820] = {X 50.2165, Y 48.3150, Z -3.0000, A 0.000, B 0.000, C 0.000 }
gfCNCPoint2[14821] = {X 49.4126, Y 48.8201, Z -3.0000, A 0.000, B 0.000, C 0.000 }
gfCNCPoint2[14822] = {X 48.5164, Y 49.1337, Z -3.0000, A 0.000, B 0.000, C 0.000 }
gfCNCPoint2[14823] = {X 47.5729, Y 49.2400, Z -3.0000, A 0.000, B 0.000, C 0.000 }
gfCNCPoint2[14824] = {X 40.6393, Y 49.2400, Z -3.0000, A 0.000, B 0.000, C 0.000 }
gfCNCPoint2[14825] = {X 39.6958, Y 49.1337, Z -3.0000, A 0.000, B 0.000, C 0.000 }
gfCNCPoint2[14826] = {X 38.7996, Y 48.8201, Z -3.0000, A 0.000, B 0.000, C 0.000 }
gfCNCPoint2[14827] = {X 37.9957, Y 48.3150, Z -3.0000, A 0.000, B 0.000, C 0.000 }
gfCNCPoint2[14828] = {X 37.3243, Y 47.6436, Z -3.0000, A 0.000, B 0.000, C 0.000 }
gfCNCPoint2[14829] = {X 36.8192, Y 46.8397, Z -3.0000, A 0.000, B 0.000, C 0.000 }
gfCNCPoint2[14830] = {X 36.5056, Y 45.9435, Z -3.0000, A 0.000, B 0.000, C 0.000 }
gfCNCPoint2[14831] = {X 36.3993, Y 45.0000, Z -3.0000, A 0.000, B 0.000, C 0.000 }
gfCNCPoint2[14832] = {X 36.3993, Y 44.2086, Z -3.0000, A 0.000, B 0.000, C 0.000 }
gfCNCPoint2[14833] = {X 36.5111, Y 43.2416, Z -3.0000, A 0.000, B 0.000, C 0.000 }
gfCNCPoint2[14834] = {X 36.8405, Y 42.3255, Z -3.0000, A 0.000, B 0.000, C 0.000 }
gfCNCPoint2[14835] = {X 37.3702, Y 41.5087, Z -3.0000, A 0.000, B 0.000, C 0.000 }
gfCNCPoint2[14836] = {X 38.0722, Y 40.8342, Z -3.0000, A 0.000, B 0.000, C 0.000 }
gfCNCPoint2[14837] = {X 38.9096, Y 40.3377, Z -3.0000, A 0.000, B 0.000, C 0.000 }
gfCNCPoint2[14838] = {X 39.0314, Y 40.2164, Z -3.0000, A 0.000, B 0.000, C 0.000 }
gfCNCPoint2[14839] = {X 39.6097, Y 38.8460, Z -3.0000, A 0.000, B 0.000, C 0.000 }
gfCNCPoint2[14840] = {X 40.1403, Y 37.4565, Z -3.0000, A 0.000, B 0.000, C 0.000 }
gfCNCPoint2[14841] = {X 43.7122, Y 27.8658, Z -3.0000, A 0.000, B 0.000, C 0.000 }
gfCNCPoint2[14842] = {X 39.9637, Y 26.4698, Z -3.0000, A 0.000, B 0.000, C 0.000 }
gfCNCPoint2[14843] = {X 43.7872, Y 27.8937, Z -3.0000, A 0.000, B 0.000, C 0.000 }
gfCNCPoint2[14844] = {X 48.4687, Y 15.3238, Z -3.0000, A 0.000, B 0.000, C 0.000 }
gfCNCPoint2[14845] = {X 48.0765, Y 14.6072, Z -3.0000, A 0.000, B 0.000, C 0.000 }
gfCNCPoint2[14846] = {X 47.8320, Y 13.8279, Z -3.0000, A 0.000, B 0.000, C 0.000 }
gfCNCPoint2[14847] = {X 47.7444, Y 13.0158, Z -3.0000, A 0.000, B 0.000, C 0.000 }
gfCNCPoint2[14848] = {X 47.7442, Y 12.1868, Z -3.0000, A 0.000, B 0.000, C 0.000 }
gfCNCPoint2[14849] = {X 47.8485, Y 11.2611, Z -3.0000, A 0.000, B 0.000, C 0.000 }
gfCNCPoint2[14850] = {X 48.1562, Y 10.3819, Z -3.0000, A 0.000, B 0.000, C 0.000 }
gfCNCPoint2[14851] = {X 48.6518, Y 9.5931, Z -3.0000, A 0.000, B 0.000, C 0.000 }
gfCNCPoint2[14852] = {X 49.3105, Y 8.9344, Z -3.0000, A 0.000, B 0.000, C 0.000 }
gfCNCPoint2[14853] = {X 50.0993, Y 8.4388, Z -3.0000, A 0.000, B 0.000, C 0.000 }
gfCNCPoint2[14854] = {X 50.9785, Y 8.1311, Z -3.0000, A 0.000, B 0.000, C 0.000 }
gfCNCPoint2[14855] = {X 51.9042, Y 8.0268, Z -3.0000, A 0.000, B 0.000, C 0.000 }
gfCNCPoint2[14856] = {X 59.6221, Y 8.0268, Z -3.0000, A 0.000, B 0.000, C 0.000 }
gfCNCPoint2[14857] = {X 60.5478, Y 8.1311, Z -3.0000, A 0.000, B 0.000, C 0.000 }
gfCNCPoint2[14858] = {X 61.4271, Y 8.4388, Z -3.0000, A 0.000, B 0.000, C 0.000 }
gfCNCPoint2[14859] = {X 62.2158, Y 8.9344, Z -3.0000, A 0.000, B 0.000, C 0.000 }
gfCNCPoint2[14860] = {X 62.8745, Y 9.5931, Z -3.0000, A 0.000, B 0.000, C 0.000 }
gfCNCPoint2[14861] = {X 63.3702, Y 10.3819, Z -3.0000, A 0.000, B 0.000, C 0.000 }
gfCNCPoint2[14862] = {X 63.6778, Y 11.2611, Z -3.0000, A 0.000, B 0.000, C 0.000 }
gfCNCPoint2[14863] = {X 63.7821, Y 12.1868, Z -3.0000, A 0.000, B 0.000, C 0.000 }
gfCNCPoint2[14864] = {X 63.7821, Y 12.9781, Z -3.0000, A 0.000, B 0.000, C 0.000 }
gfCNCPoint2[14865] = {X 63.6960, Y 13.8204, Z -3.0000, A 0.000, B 0.000, C 0.000 }
gfCNCPoint2[14866] = {X 63.4410, Y 14.6277, Z -3.0000, A 0.000, B 0.000, C 0.000 }
gfCNCPoint2[14867] = {X 63.0280, Y 15.3667, Z -3.0000, A 0.000, B 0.000, C 0.000 }
gfCNCPoint2[14868] = {X 63.2755, Y 16.0199, Z -3.0000, A 0.000, B 0.000, C 0.000 }
gfCNCPoint2[14869] = {X 65.8846, Y 22.9435, Z -3.0000, A 0.000, B 0.000, C 0.000 }
gfCNCPoint2[14870] = {X 72.0597, Y 39.5578, Z -3.0000, A 0.000, B 0.000, C 0.000 }
gfCNCPoint2[14871] = {X 72.3897, Y 40.3880, Z -3.0000, A 0.000, B 0.000, C 0.000 }
gfCNCPoint2[14872] = {X 73.2208, Y 40.8661, Z -3.0000, A 0.000, B 0.000, C 0.000 }
gfCNCPoint2[14873] = {X 73.9203, Y 41.5219, Z -3.0000, A 0.000, B 0.000, C 0.000 }
gfCNCPoint2[14874] = {X 74.4512, Y 42.3204, Z -3.0000, A 0.000, B 0.000, C 0.000 }
gfCNCPoint2[14875] = {X 74.7850, Y 43.2192, Z -3.0000, A 0.000, B 0.000, C 0.000 }
gfCNCPoint2[14876] = {X 74.9043, Y 44.1706, Z -3.0000, A 0.000, B 0.000, C 0.000 }
gfCNCPoint2[14877] = {X 74.9045, Y 45.0000, Z -3.0000, A 0.000, B 0.000, C 0.000 }
gfCNCPoint2[14878] = {X 74.8002, Y 45.9257, Z -3.0000, A 0.000, B 0.000, C 0.000 }
gfCNCPoint2[14879] = {X 74.4925, Y 46.8050, Z -3.0000, A 0.000, B 0.000, C 0.000 }
gfCNCPoint2[14880] = {X 73.9969, Y 47.5937, Z -3.0000, A 0.000, B 0.000, C 0.000 }
gfCNCPoint2[14881] = {X 73.3382, Y 48.2524, Z -3.0000, A 0.000, B 0.000, C 0.000 }
gfCNCPoint2[14882] = {X 72.5494, Y 48.7480, Z -3.0000, A 0.000, B 0.000, C 0.000 }
gfCNCPoint2[14883] = {X 71.6701, Y 49.0557, Z -3.0000, A 0.000, B 0.000, C 0.000 }
gfCNCPoint2[14884] = {X 70.7445, Y 49.1600, Z -3.0000, A 0.000, B 0.000, C 0.000 }
gfCNCPoint2[14885] = {X 64.1851, Y 49.1600, Z -3.0000, A 0.000, B 0.000, C 0.000 }
gfCNCPoint2[14886] = {X 63.2594, Y 49.0557, Z -3.0000, A 0.000, B 0.000, C 0.000 }
gfCNCPoint2[14887] = {X 62.3802, Y 48.7480, Z -3.0000, A 0.000, B 0.000, C 0.000 }
gfCNCPoint2[14888] = {X 61.5914, Y 48.2524, Z -3.0000, A 0.000, B 0.000, C 0.000 }
gfCNCPoint2[14889] = {X 60.9327, Y 47.5937, Z -3.0000, A 0.000, B 0.000, C 0.000 }
gfCNCPoint2[14890] = {X 60.4371, Y 46.8050, Z -3.0000, A 0.000, B 0.000, C 0.000 }
gfCNCPoint2[14891] = {X 60.1294, Y 45.9257, Z -3.0000, A 0.000, B 0.000, C 0.000 }
gfCNCPoint2[14892] = {X 60.0251, Y 45.0000, Z -3.0000, A 0.000, B 0.000, C 0.000 }
gfCNCPoint2[14893] = {X 60.0251, Y 44.2086, Z -3.0000, A 0.000, B 0.000, C 0.000 }
gfCNCPoint2[14894] = {X 60.1143, Y 43.3552, Z -3.0000, A 0.000, B 0.000, C 0.000 }
gfCNCPoint2[14895] = {X 60.3767, Y 42.5383, Z -3.0000, A 0.000, B 0.000, C 0.000 }
gfCNCPoint2[14896] = {X 60.8011, Y 41.7925, Z -3.0000, A 0.000, B 0.000, C 0.000 }
gfCNCPoint2[14897] = {X 60.1190, Y 39.9292, Z -3.0000, A 0.000, B 0.000, C 0.000 }
gfCNCPoint2[14898] = {X 51.9656, Y 39.9292, Z -3.0000, A 0.000, B 0.000, C 0.000 }
gfCNCPoint2[14899] = {X 51.1572, Y 42.1008, Z -3.0000, A 0.000, B 0.000, C 0.000 }
gfCNCPoint2[14900] = {X 51.1991, Y 42.1700, Z -3.0000, A 0.000, B 0.000, C 0.000 }
gfCNCPoint2[14901] = {X 51.4888, Y 42.8046, Z -3.0000, A 0.000, B 0.000, C 0.000 }
gfCNCPoint2[14902] = {X 51.6684, Y 43.4787, Z -3.0000, A 0.000, B 0.000, C 0.000 }
gfCNCPoint2[14903] = {X 51.7328, Y 44.1733, Z -3.0000, A 0.000, B 0.000, C 0.000 }
gfCNCPoint2[14904] = {X 51.7329, Y 45.0000, Z -3.0000, A 0.000, B 0.000, C 0.000 }
gfCNCPoint2[14905] = {X 51.6286, Y 45.9257, Z -3.0000, A 0.000, B 0.000, C 0.000 }
gfCNCPoint2[14906] = {X 51.3210, Y 46.8050, Z -3.0000, A 0.000, B 0.000, C 0.000 }
gfCNCPoint2[14907] = {X 50.8253, Y 47.5937, Z -3.0000, A 0.000, B 0.000, C 0.000 }
gfCNCPoint2[14908] = {X 50.1666, Y 48.2524, Z -3.0000, A 0.000, B 0.000, C 0.000 }
gfCNCPoint2[14909] = {X 49.3779, Y 48.7480, Z -3.0000, A 0.000, B 0.000, C 0.000 }
gfCNCPoint2[14910] = {X 48.4986, Y 49.0557, Z -3.0000, A 0.000, B 0.000, C 0.000 }
gfCNCPoint2[14911] = {X 47.5729, Y 49.1600, Z -3.0000, A 0.000, B 0.000, C 0.000 }
gfCNCPoint2[14912] = {X 40.6393, Y 49.1600, Z -3.0000, A 0.000, B 0.000, C 0.000 }
gfCNCPoint2[14913] = {X 39.7136, Y 49.0557, Z -3.0000, A 0.000, B 0.000, C 0.000 }
gfCNCPoint2[14914] = {X 38.8343, Y 48.7480, Z -3.0000, A 0.000, B 0.000, C 0.000 }
gfCNCPoint2[14915] = {X 38.0456, Y 48.2524, Z -3.0000, A 0.000, B 0.000, C 0.000 }
gfCNCPoint2[14916] = {X 37.3869, Y 47.5937, Z -3.0000, A 0.000, B 0.000, C 0.000 }
gfCNCPoint2[14917] = {X 36.8913, Y 46.8050, Z -3.0000, A 0.000, B 0.000, C 0.000 }
gfCNCPoint2[14918] = {X 36.5836, Y 45.9257, Z -3.0000, A 0.000, B 0.000, C 0.000 }
gfCNCPoint2[14919] = {X 36.4793, Y 45.0000, Z -3.0000, A 0.000, B 0.000, C 0.000 }
gfCNCPoint2[14920] = {X 36.4793, Y 44.2086, Z -3.0000, A 0.000, B 0.000, C 0.000 }
gfCNCPoint2[14921] = {X 36.5897, Y 43.2570, Z -3.0000, A 0.000, B 0.000, C 0.000 }
gfCNCPoint2[14922] = {X 36.9148, Y 42.3558, Z -3.0000, A 0.000, B 0.000, C 0.000 }
gfCNCPoint2[14923] = {X 37.4375, Y 41.5529, Z -3.0000, A 0.000, B 0.000, C 0.000 }
gfCNCPoint2[14924] = {X 38.1300, Y 40.8908, Z -3.0000, A 0.000, B 0.000, C 0.000 }
gfCNCPoint2[14925] = {X 38.9556, Y 40.4048, Z -3.0000, A 0.000, B 0.000, C 0.000 }
gfCNCPoint2[14926] = {X 39.0985, Y 40.2625, Z -3.0000, A 0.000, B 0.000, C 0.000 }
gfCNCPoint2[14927] = {X 39.6811, Y 38.8828, Z -3.0000, A 0.000, B 0.000, C 0.000 }
gfCNCPoint2[14928] = {X 40.2155, Y 37.4838, Z -3.0000, A 0.000, B 0.000, C 0.000 }
gfCNCPoint2[14929] = {X 43.7872, Y 27.8937, Z -3.0000, A 0.000, B 0.000, C 0.000 }
gfCNCPoint2[14930] = {X 40.0387, Y 26.4977, Z -3.0000, A 0.000, B 0.000, C 0.000 }
gfCNCPoint2[14931] = {X 43.8621, Y 27.9217, Z -3.0000, A 0.000, B 0.000, C 0.000 }
gfCNCPoint2[14932] = {X 48.5582, Y 15.3126, Z -3.0000, A 0.000, B 0.000, C 0.000 }
gfCNCPoint2[14933] = {X 48.1610, Y 14.6012, Z -3.0000, A 0.000, B 0.000, C 0.000 }
gfCNCPoint2[14934] = {X 47.9131, Y 13.8250, Z -3.0000, A 0.000, B 0.000, C 0.000 }
gfCNCPoint2[14935] = {X 47.8244, Y 13.0151, Z -3.0000, A 0.000, B 0.000, C 0.000 }
gfCNCPoint2[14936] = {X 47.8242, Y 12.1868, Z -3.0000, A 0.000, B 0.000, C 0.000 }
gfCNCPoint2[14937] = {X 47.9265, Y 11.2789, Z -3.0000, A 0.000, B 0.000, C 0.000 }
gfCNCPoint2[14938] = {X 48.2283, Y 10.4166, Z -3.0000, A 0.000, B 0.000, C 0.000 }
gfCNCPoint2[14939] = {X 48.7144, Y 9.6430, Z -3.0000, A 0.000, B 0.000, C 0.000 }
gfCNCPoint2[14940] = {X 49.3604, Y 8.9969, Z -3.0000, A 0.000, B 0.000, C 0.000 }
gfCNCPoint2[14941] = {X 50.1340, Y 8.5109, Z -3.0000, A 0.000, B 0.000, C 0.000 }
gfCNCPoint2[14942] = {X 50.9963, Y 8.2091, Z -3.0000, A 0.000, B 0.000, C 0.000 }
gfCNCPoint2[14943] = {X 51.9042, Y 8.1068, Z -3.0000, A 0.000, B 0.000, C 0.000 }
gfCNCPoint2[14944] = {X 59.6221, Y 8.1068, Z -3.0000, A 0.000, B 0.000, C 0.000 }
gfCNCPoint2[14945] = {X 60.5300, Y 8.2091, Z -3.0000, A 0.000, B 0.000, C 0.000 }
gfCNCPoint2[14946] = {X 61.3924, Y 8.5109, Z -3.0000, A 0.000, B 0.000, C 0.000 }
gfCNCPoint2[14947] = {X 62.1660, Y 8.9969, Z -3.0000, A 0.000, B 0.000, C 0.000 }
gfCNCPoint2[14948] = {X 62.8120, Y 9.6430, Z -3.0000, A 0.000, B 0.000, C 0.000 }
gfCNCPoint2[14949] = {X 63.2981, Y 10.4166, Z -3.0000, A 0.000, B 0.000, C 0.000 }
gfCNCPoint2[14950] = {X 63.5998, Y 11.2789, Z -3.0000, A 0.000, B 0.000, C 0.000 }
gfCNCPoint2[14951] = {X 63.7021, Y 12.1868, Z -3.0000, A 0.000, B 0.000, C 0.000 }
gfCNCPoint2[14952] = {X 63.7021, Y 12.9781, Z -3.0000, A 0.000, B 0.000, C 0.000 }
gfCNCPoint2[14953] = {X 63.6147, Y 13.8179, Z -3.0000, A 0.000, B 0.000, C 0.000 }
gfCNCPoint2[14954] = {X 63.3564, Y 14.6218, Z -3.0000, A 0.000, B 0.000, C 0.000 }
gfCNCPoint2[14955] = {X 62.9381, Y 15.3552, Z -3.0000, A 0.000, B 0.000, C 0.000 }
gfCNCPoint2[14956] = {X 63.2006, Y 16.0481, Z -3.0000, A 0.000, B 0.000, C 0.000 }
gfCNCPoint2[14957] = {X 65.8097, Y 22.9716, Z -3.0000, A 0.000, B 0.000, C 0.000 }
gfCNCPoint2[14958] = {X 71.9850, Y 39.5865, Z -3.0000, A 0.000, B 0.000, C 0.000 }
gfCNCPoint2[14959] = {X 72.3277, Y 40.4485, Z -3.0000, A 0.000, B 0.000, C 0.000 }
gfCNCPoint2[14960] = {X 73.1519, Y 40.9148, Z -3.0000, A 0.000, B 0.000, C 0.000 }
gfCNCPoint2[14961] = {X 73.8464, Y 41.5585, Z -3.0000, A 0.000, B 0.000, C 0.000 }
gfCNCPoint2[14962] = {X 74.3739, Y 42.3450, Z -3.0000, A 0.000, B 0.000, C 0.000 }
gfCNCPoint2[14963] = {X 74.7058, Y 43.2318, Z -3.0000, A 0.000, B 0.000, C 0.000 }
gfCNCPoint2[14964] = {X 74.8243, Y 44.1714, Z -3.0000, A 0.000, B 0.000, C 0.000 }
gfCNCPoint2[14965] = {X 74.8245, Y 45.0000, Z -3.0000, A 0.000, B 0.000, C 0.000 }
gfCNCPoint2[14966] = {X 74.7222, Y 45.9079, Z -3.0000, A 0.000, B 0.000, C 0.000 }
gfCNCPoint2[14967] = {X 74.4204, Y 46.7702, Z -3.0000, A 0.000, B 0.000, C 0.000 }
gfCNCPoint2[14968] = {X 73.9343, Y 47.5438, Z -3.0000, A 0.000, B 0.000, C 0.000 }
gfCNCPoint2[14969] = {X 73.2883, Y 48.1899, Z -3.0000, A 0.000, B 0.000, C 0.000 }
gfCNCPoint2[14970] = {X 72.5147, Y 48.6760, Z -3.0000, A 0.000, B 0.000, C 0.000 }
gfCNCPoint2[14971] = {X 71.6523, Y 48.9777, Z -3.0000, A 0.000, B 0.000, C 0.000 }
gfCNCPoint2[14972] = {X 70.7445, Y 49.0800, Z -3.0000, A 0.000, B 0.000, C 0.000 }
gfCNCPoint2[14973] = {X 64.1851, Y 49.0800, Z -3.0000, A 0.000, B 0.000, C 0.000 }
gfCNCPoint2[14974] = {X 63.2772, Y 48.9777, Z -3.0000, A 0.000, B 0.000, C 0.000 }
gfCNCPoint2[14975] = {X 62.4149, Y 48.6760, Z -3.0000, A 0.000, B 0.000, C 0.000 }
gfCNCPoint2[14976] = {X 61.6413, Y 48.1899, Z -3.0000, A 0.000, B 0.000, C 0.000 }
gfCNCPoint2[14977] = {X 60.9953, Y 47.5438, Z -3.0000, A 0.000, B 0.000, C 0.000 }
gfCNCPoint2[14978] = {X 60.5092, Y 46.7702, Z -3.0000, A 0.000, B 0.000, C 0.000 }
gfCNCPoint2[14979] = {X 60.2074, Y 45.9079, Z -3.0000, A 0.000, B 0.000, C 0.000 }
gfCNCPoint2[14980] = {X 60.1051, Y 45.0000, Z -3.0000, A 0.000, B 0.000, C 0.000 }
gfCNCPoint2[14981] = {X 60.1051, Y 44.2086, Z -3.0000, A 0.000, B 0.000, C 0.000 }
gfCNCPoint2[14982] = {X 60.1955, Y 43.3579, Z -3.0000, A 0.000, B 0.000, C 0.000 }
gfCNCPoint2[14983] = {X 60.4613, Y 42.5448, Z -3.0000, A 0.000, B 0.000, C 0.000 }
gfCNCPoint2[14984] = {X 60.8908, Y 41.8049, Z -3.0000, A 0.000, B 0.000, C 0.000 }
gfCNCPoint2[14985] = {X 60.1749, Y 39.8492, Z -3.0000, A 0.000, B 0.000, C 0.000 }
gfCNCPoint2[14986] = {X 51.9100, Y 39.8492, Z -3.0000, A 0.000, B 0.000, C 0.000 }
gfCNCPoint2[14987] = {X 51.0687, Y 42.1091, Z -3.0000, A 0.000, B 0.000, C 0.000 }
gfCNCPoint2[14988] = {X 51.1306, Y 42.2115, Z -3.0000, A 0.000, B 0.000, C 0.000 }
gfCNCPoint2[14989] = {X 51.4141, Y 42.8332, Z -3.0000, A 0.000, B 0.000, C 0.000 }
gfCNCPoint2[14990] = {X 51.5898, Y 43.4936, Z -3.0000, A 0.000, B 0.000, C 0.000 }
gfCNCPoint2[14991] = {X 51.6528, Y 44.1740, Z -3.0000, A 0.000, B 0.000, C 0.000 }
gfCNCPoint2[14992] = {X 51.6529, Y 45.0000, Z -3.0000, A 0.000, B 0.000, C 0.000 }
gfCNCPoint2[14993] = {X 51.5506, Y 45.9079, Z -3.0000, A 0.000, B 0.000, C 0.000 }
gfCNCPoint2[14994] = {X 51.2489, Y 46.7702, Z -3.0000, A 0.000, B 0.000, C 0.000 }
gfCNCPoint2[14995] = {X 50.7628, Y 47.5438, Z -3.0000, A 0.000, B 0.000, C 0.000 }
gfCNCPoint2[14996] = {X 50.1168, Y 48.1899, Z -3.0000, A 0.000, B 0.000, C 0.000 }
gfCNCPoint2[14997] = {X 49.3432, Y 48.6760, Z -3.0000, A 0.000, B 0.000, C 0.000 }
gfCNCPoint2[14998] = {X 48.4808, Y 48.9777, Z -3.0000, A 0.000, B 0.000, C 0.000 }
gfCNCPoint2[14999] = {X 47.5729, Y 49.0800, Z -3.0000, A 0.000, B 0.000, C 0.000 }
gfCNCPoint2[15000] = {X 40.6393, Y 49.0800, Z -3.0000, A 0.000, B 0.000, C 0.000 }
gfCNCPoint2[15001] = {X 39.7314, Y 48.9777, Z -3.0000, A 0.000, B 0.000, C 0.000 }
gfCNCPoint2[15002] = {X 38.8691, Y 48.6760, Z -3.0000, A 0.000, B 0.000, C 0.000 }
gfCNCPoint2[15003] = {X 38.0955, Y 48.1899, Z -3.0000, A 0.000, B 0.000, C 0.000 }
gfCNCPoint2[15004] = {X 37.4494, Y 47.5438, Z -3.0000, A 0.000, B 0.000, C 0.000 }
gfCNCPoint2[15005] = {X 36.9633, Y 46.7702, Z -3.0000, A 0.000, B 0.000, C 0.000 }
gfCNCPoint2[15006] = {X 36.6616, Y 45.9079, Z -3.0000, A 0.000, B 0.000, C 0.000 }
gfCNCPoint2[15007] = {X 36.5593, Y 45.0000, Z -3.0000, A 0.000, B 0.000, C 0.000 }
gfCNCPoint2[15008] = {X 36.5593, Y 44.2086, Z -3.0000, A 0.000, B 0.000, C 0.000 }
gfCNCPoint2[15009] = {X 36.6682, Y 43.2724, Z -3.0000, A 0.000, B 0.000, C 0.000 }
gfCNCPoint2[15010] = {X 36.9891, Y 42.3861, Z -3.0000, A 0.000, B 0.000, C 0.000 }
gfCNCPoint2[15011] = {X 37.5047, Y 41.5971, Z -3.0000, A 0.000, B 0.000, C 0.000 }
gfCNCPoint2[15012] = {X 38.1877, Y 40.9475, Z -3.0000, A 0.000, B 0.000, C 0.000 }
gfCNCPoint2[15013] = {X 39.0014, Y 40.4720, Z -3.0000, A 0.000, B 0.000, C 0.000 }
gfCNCPoint2[15014] = {X 39.1655, Y 40.3086, Z -3.0000, A 0.000, B 0.000, C 0.000 }
gfCNCPoint2[15015] = {X 39.7525, Y 38.9196, Z -3.0000, A 0.000, B 0.000, C 0.000 }
gfCNCPoint2[15016] = {X 40.2907, Y 37.5110, Z -3.0000, A 0.000, B 0.000, C 0.000 }
gfCNCPoint2[15017] = {X 43.8621, Y 27.9217, Z -3.0000, A 0.000, B 0.000, C 0.000 }
gfCNCPoint2[15018] = {X 40.1137, Y 26.5256, Z -3.0000, A 0.000, B 0.000, C 0.000 }
gfCNCPoint2[15019] = {X 43.9371, Y 27.9496, Z -3.0000, A 0.000, B 0.000, C 0.000 }
gfCNCPoint2[15020] = {X 48.6479, Y 15.3010, Z -3.0000, A 0.000, B 0.000, C 0.000 }
gfCNCPoint2[15021] = {X 48.2407, Y 14.5838, Z -3.0000, A 0.000, B 0.000, C 0.000 }
gfCNCPoint2[15022] = {X 47.9892, Y 13.7983, Z -3.0000, A 0.000, B 0.000, C 0.000 }
gfCNCPoint2[15023] = {X 47.9042, Y 12.9779, Z -3.0000, A 0.000, B 0.000, C 0.000 }
gfCNCPoint2[15024] = {X 47.9042, Y 12.1868, Z -3.0000, A 0.000, B 0.000, C 0.000 }
gfCNCPoint2[15025] = {X 48.0045, Y 11.2967, Z -3.0000, A 0.000, B 0.000, C 0.000 }
gfCNCPoint2[15026] = {X 48.3003, Y 10.4513, Z -3.0000, A 0.000, B 0.000, C 0.000 }
gfCNCPoint2[15027] = {X 48.7769, Y 9.6929, Z -3.0000, A 0.000, B 0.000, C 0.000 }
gfCNCPoint2[15028] = {X 49.4103, Y 9.0595, Z -3.0000, A 0.000, B 0.000, C 0.000 }
gfCNCPoint2[15029] = {X 50.1687, Y 8.5829, Z -3.0000, A 0.000, B 0.000, C 0.000 }
gfCNCPoint2[15030] = {X 51.0141, Y 8.2871, Z -3.0000, A 0.000, B 0.000, C 0.000 }
gfCNCPoint2[15031] = {X 51.9042, Y 8.1868, Z -3.0000, A 0.000, B 0.000, C 0.000 }
gfCNCPoint2[15032] = {X 59.6221, Y 8.1868, Z -3.0000, A 0.000, B 0.000, C 0.000 }
gfCNCPoint2[15033] = {X 60.5122, Y 8.2871, Z -3.0000, A 0.000, B 0.000, C 0.000 }
gfCNCPoint2[15034] = {X 61.3577, Y 8.5829, Z -3.0000, A 0.000, B 0.000, C 0.000 }
gfCNCPoint2[15035] = {X 62.1161, Y 9.0595, Z -3.0000, A 0.000, B 0.000, C 0.000 }
gfCNCPoint2[15036] = {X 62.7495, Y 9.6929, Z -3.0000, A 0.000, B 0.000, C 0.000 }
gfCNCPoint2[15037] = {X 63.2260, Y 10.4513, Z -3.0000, A 0.000, B 0.000, C 0.000 }
gfCNCPoint2[15038] = {X 63.5218, Y 11.2967, Z -3.0000, A 0.000, B 0.000, C 0.000 }
gfCNCPoint2[15039] = {X 63.6221, Y 12.1868, Z -3.0000, A 0.000, B 0.000, C 0.000 }
gfCNCPoint2[15040] = {X 63.6219, Y 13.0192, Z -3.0000, A 0.000, B 0.000, C 0.000 }
gfCNCPoint2[15041] = {X 63.5277, Y 13.8422, Z -3.0000, A 0.000, B 0.000, C 0.000 }
gfCNCPoint2[15042] = {X 63.2659, Y 14.6281, Z -3.0000, A 0.000, B 0.000, C 0.000 }
gfCNCPoint2[15043] = {X 62.8480, Y 15.3432, Z -3.0000, A 0.000, B 0.000, C 0.000 }
gfCNCPoint2[15044] = {X 63.1258, Y 16.0764, Z -3.0000, A 0.000, B 0.000, C 0.000 }
gfCNCPoint2[15045] = {X 65.7348, Y 22.9996, Z -3.0000, A 0.000, B 0.000, C 0.000 }
gfCNCPoint2[15046] = {X 71.9103, Y 39.6152, Z -3.0000, A 0.000, B 0.000, C 0.000 }
gfCNCPoint2[15047] = {X 72.2609, Y 40.4970, Z -3.0000, A 0.000, B 0.000, C 0.000 }
gfCNCPoint2[15048] = {X 72.2781, Y 40.5145, Z -3.0000, A 0.000, B 0.000, C 0.000 }
gfCNCPoint2[15049] = {X 72.3443, Y 40.5427, Z -3.0000, A 0.000, B 0.000, C 0.000 }
gfCNCPoint2[15050] = {X 72.4100, Y 40.5720, Z -3.0000, A 0.000, B 0.000, C 0.000 }
gfCNCPoint2[15051] = {X 73.1898, Y 41.0433, Z -3.0000, A 0.000, B 0.000, C 0.000 }
gfCNCPoint2[15052] = {X 73.8427, Y 41.6788, Z -3.0000, A 0.000, B 0.000, C 0.000 }
gfCNCPoint2[15053] = {X 74.3348, Y 42.4455, Z -3.0000, A 0.000, B 0.000, C 0.000 }
gfCNCPoint2[15054] = {X 74.6407, Y 43.3037, Z -3.0000, A 0.000, B 0.000, C 0.000 }
gfCNCPoint2[15055] = {X 74.7445, Y 44.2089, Z -3.0000, A 0.000, B 0.000, C 0.000 }
gfCNCPoint2[15056] = {X 74.7445, Y 45.0000, Z -3.0000, A 0.000, B 0.000, C 0.000 }
gfCNCPoint2[15057] = {X 74.6442, Y 45.8901, Z -3.0000, A 0.000, B 0.000, C 0.000 }
gfCNCPoint2[15058] = {X 74.3483, Y 46.7355, Z -3.0000, A 0.000, B 0.000, C 0.000 }
gfCNCPoint2[15059] = {X 73.8718, Y 47.4940, Z -3.0000, A 0.000, B 0.000, C 0.000 }
gfCNCPoint2[15060] = {X 73.2384, Y 48.1273, Z -3.0000, A 0.000, B 0.000, C 0.000 }
gfCNCPoint2[15061] = {X 72.4800, Y 48.6039, Z -3.0000, A 0.000, B 0.000, C 0.000 }
gfCNCPoint2[15062] = {X 71.6345, Y 48.8997, Z -3.0000, A 0.000, B 0.000, C 0.000 }
gfCNCPoint2[15063] = {X 70.7445, Y 49.0000, Z -3.0000, A 0.000, B 0.000, C 0.000 }
gfCNCPoint2[15064] = {X 64.1851, Y 49.0000, Z -3.0000, A 0.000, B 0.000, C 0.000 }
gfCNCPoint2[15065] = {X 63.2951, Y 48.8997, Z -3.0000, A 0.000, B 0.000, C 0.000 }
gfCNCPoint2[15066] = {X 62.4496, Y 48.6039, Z -3.0000, A 0.000, B 0.000, C 0.000 }
gfCNCPoint2[15067] = {X 61.6912, Y 48.1273, Z -3.0000, A 0.000, B 0.000, C 0.000 }
gfCNCPoint2[15068] = {X 61.0578, Y 47.4940, Z -3.0000, A 0.000, B 0.000, C 0.000 }
gfCNCPoint2[15069] = {X 60.5813, Y 46.7355, Z -3.0000, A 0.000, B 0.000, C 0.000 }
gfCNCPoint2[15070] = {X 60.2854, Y 45.8901, Z -3.0000, A 0.000, B 0.000, C 0.000 }
gfCNCPoint2[15071] = {X 60.1851, Y 45.0000, Z -3.0000, A 0.000, B 0.000, C 0.000 }
gfCNCPoint2[15072] = {X 60.1855, Y 44.1538, Z -3.0000, A 0.000, B 0.000, C 0.000 }
gfCNCPoint2[15073] = {X 60.2746, Y 43.3674, Z -3.0000, A 0.000, B 0.000, C 0.000 }
gfCNCPoint2[15074] = {X 60.5168, Y 42.6140, Z -3.0000, A 0.000, B 0.000, C 0.000 }
gfCNCPoint2[15075] = {X 60.9025, Y 41.9231, Z -3.0000, A 0.000, B 0.000, C 0.000 }
gfCNCPoint2[15076] = {X 60.9808, Y 41.8181, Z -3.0000, A 0.000, B 0.000, C 0.000 }
gfCNCPoint2[15077] = {X 60.2308, Y 39.7692, Z -3.0000, A 0.000, B 0.000, C 0.000 }
gfCNCPoint2[15078] = {X 51.8421, Y 39.7692, Z -3.0000, A 0.000, B 0.000, C 0.000 }
gfCNCPoint2[15079] = {X 51.8421, Y 39.8024, Z -3.0000, A 0.000, B 0.000, C 0.000 }
gfCNCPoint2[15080] = {X 50.9803, Y 42.1175, Z -3.0000, A 0.000, B 0.000, C 0.000 }
gfCNCPoint2[15081] = {X 51.0722, Y 42.2709, Z -3.0000, A 0.000, B 0.000, C 0.000 }
gfCNCPoint2[15082] = {X 51.3477, Y 42.8856, Z -3.0000, A 0.000, B 0.000, C 0.000 }
gfCNCPoint2[15083] = {X 51.5162, Y 43.5377, Z -3.0000, A 0.000, B 0.000, C 0.000 }
gfCNCPoint2[15084] = {X 51.5729, Y 44.2089, Z -3.0000, A 0.000, B 0.000, C 0.000 }
gfCNCPoint2[15085] = {X 51.5729, Y 45.0000, Z -3.0000, A 0.000, B 0.000, C 0.000 }
gfCNCPoint2[15086] = {X 51.4726, Y 45.8901, Z -3.0000, A 0.000, B 0.000, C 0.000 }
gfCNCPoint2[15087] = {X 51.1768, Y 46.7355, Z -3.0000, A 0.000, B 0.000, C 0.000 }
gfCNCPoint2[15088] = {X 50.7003, Y 47.4940, Z -3.0000, A 0.000, B 0.000, C 0.000 }
gfCNCPoint2[15089] = {X 50.0669, Y 48.1273, Z -3.0000, A 0.000, B 0.000, C 0.000 }
gfCNCPoint2[15090] = {X 49.3085, Y 48.6039, Z -3.0000, A 0.000, B 0.000, C 0.000 }
gfCNCPoint2[15091] = {X 48.4630, Y 48.8997, Z -3.0000, A 0.000, B 0.000, C 0.000 }
gfCNCPoint2[15092] = {X 47.5729, Y 49.0000, Z -3.0000, A 0.000, B 0.000, C 0.000 }
gfCNCPoint2[15093] = {X 40.6393, Y 49.0000, Z -3.0000, A 0.000, B 0.000, C 0.000 }
gfCNCPoint2[15094] = {X 39.7492, Y 48.8997, Z -3.0000, A 0.000, B 0.000, C 0.000 }
gfCNCPoint2[15095] = {X 38.9038, Y 48.6039, Z -3.0000, A 0.000, B 0.000, C 0.000 }
gfCNCPoint2[15096] = {X 38.1453, Y 48.1273, Z -3.0000, A 0.000, B 0.000, C 0.000 }
gfCNCPoint2[15097] = {X 37.5120, Y 47.4940, Z -3.0000, A 0.000, B 0.000, C 0.000 }
gfCNCPoint2[15098] = {X 37.0354, Y 46.7355, Z -3.0000, A 0.000, B 0.000, C 0.000 }
gfCNCPoint2[15099] = {X 36.7396, Y 45.8901, Z -3.0000, A 0.000, B 0.000, C 0.000 }
gfCNCPoint2[15100] = {X 36.6393, Y 45.0000, Z -3.0000, A 0.000, B 0.000, C 0.000 }
gfCNCPoint2[15101] = {X 36.6397, Y 44.1538, Z -3.0000, A 0.000, B 0.000, C 0.000 }
gfCNCPoint2[15102] = {X 36.7564, Y 43.2481, Z -3.0000, A 0.000, B 0.000, C 0.000 }
gfCNCPoint2[15103] = {X 37.0755, Y 42.3925, Z -3.0000, A 0.000, B 0.000, C 0.000 }
gfCNCPoint2[15104] = {X 37.5803, Y 41.6315, Z -3.0000, A 0.000, B 0.000, C 0.000 }
gfCNCPoint2[15105] = {X 38.2445, Y 41.0049, Z -3.0000, A 0.000, B 0.000, C 0.000 }
gfCNCPoint2[15106] = {X 39.0336, Y 40.5452, Z -3.0000, A 0.000, B 0.000, C 0.000 }
gfCNCPoint2[15107] = {X 39.0871, Y 40.5222, Z -3.0000, A 0.000, B 0.000, C 0.000 }
gfCNCPoint2[15108] = {X 39.1410, Y 40.5000, Z -3.0000, A 0.000, B 0.000, C 0.000 }
gfCNCPoint2[15109] = {X 39.1690, Y 40.4818, Z -3.0000, A 0.000, B 0.000, C 0.000 }
gfCNCPoint2[15110] = {X 39.1881, Y 40.4545, Z -3.0000, A 0.000, B 0.000, C 0.000 }
gfCNCPoint2[15111] = {X 39.2134, Y 40.3978, Z -3.0000, A 0.000, B 0.000, C 0.000 }
gfCNCPoint2[15112] = {X 39.2387, Y 40.3410, Z -3.0000, A 0.000, B 0.000, C 0.000 }
gfCNCPoint2[15113] = {X 39.8267, Y 38.9495, Z -3.0000, A 0.000, B 0.000, C 0.000 }
gfCNCPoint2[15114] = {X 40.3659, Y 37.5383, Z -3.0000, A 0.000, B 0.000, C 0.000 }
gfCNCPoint2[15115] = {X 43.9371, Y 27.9496, Z -3.0000, A 0.000, B 0.000, C 0.000 }
gfCNCPoint2[15116] = {X 40.1137, Y 26.5256, Z -3.0000, A 0.000, B 0.000, C 0.000 }
gfCNCPoint2[15117] = {X 40.1137, Y 26.5256, Z 0.0000, A 0.000, B 0.000, C 0.000 }
gfCNCPoint2[15118] = {X 40.1137, Y 26.5256, Z 11.0000, A 0.000, B 0.000, C 0.000 }
gfCNCPoint2[15119] = {X 79.0233, Y 28.5920, Z 11.0000, A 0.000, B 0.000, C 0.000 }
gfCNCPoint2[15120] = {X 79.0233, Y 28.5920, Z 0.0000, A 0.000, B 0.000, C 0.000 }
gfCNCPoint2[15121] = {X 79.0233, Y 28.5920, Z -3.0000, A 0.000, B 0.000, C 0.000 }
gfCNCPoint2[15122] = {X 83.1033, Y 28.5920, Z -3.0000, A 0.000, B 0.000, C 0.000 }
gfCNCPoint2[15123] = {X 83.1031, Y 16.2746, Z -3.0000, A 0.000, B 0.000, C 0.000 }
gfCNCPoint2[15124] = {X 82.4644, Y 15.6034, Z -3.0000, A 0.000, B 0.000, C 0.000 }
gfCNCPoint2[15125] = {X 81.9834, Y 14.8115, Z -3.0000, A 0.000, B 0.000, C 0.000 }
gfCNCPoint2[15126] = {X 81.6824, Y 13.9352, Z -3.0000, A 0.000, B 0.000, C 0.000 }
gfCNCPoint2[15127] = {X 81.5752, Y 13.0148, Z -3.0000, A 0.000, B 0.000, C 0.000 }
gfCNCPoint2[15128] = {X 81.5751, Y 12.1868, Z -3.0000, A 0.000, B 0.000, C 0.000 }
gfCNCPoint2[15129] = {X 81.6834, Y 11.2255, Z -3.0000, A 0.000, B 0.000, C 0.000 }
gfCNCPoint2[15130] = {X 82.0029, Y 10.3124, Z -3.0000, A 0.000, B 0.000, C 0.000 }
gfCNCPoint2[15131] = {X 82.5176, Y 9.4933, Z -3.0000, A 0.000, B 0.000, C 0.000 }
gfCNCPoint2[15132] = {X 83.2016, Y 8.8093, Z -3.0000, A 0.000, B 0.000, C 0.000 }
gfCNCPoint2[15133] = {X 84.0207, Y 8.2946, Z -3.0000, A 0.000, B 0.000, C 0.000 }
gfCNCPoint2[15134] = {X 84.9338, Y 7.9751, Z -3.0000, A 0.000, B 0.000, C 0.000 }
gfCNCPoint2[15135] = {X 85.8951, Y 7.8668, Z -3.0000, A 0.000, B 0.000, C 0.000 }
gfCNCPoint2[15136] = {X 94.0497, Y 7.8668, Z -3.0000, A 0.000, B 0.000, C 0.000 }
gfCNCPoint2[15137] = {X 95.0110, Y 7.9751, Z -3.0000, A 0.000, B 0.000, C 0.000 }
gfCNCPoint2[15138] = {X 95.9240, Y 8.2946, Z -3.0000, A 0.000, B 0.000, C 0.000 }
gfCNCPoint2[15139] = {X 96.7431, Y 8.8093, Z -3.0000, A 0.000, B 0.000, C 0.000 }
gfCNCPoint2[15140] = {X 97.4272, Y 9.4933, Z -3.0000, A 0.000, B 0.000, C 0.000 }
gfCNCPoint2[15141] = {X 97.9419, Y 10.3124, Z -3.0000, A 0.000, B 0.000, C 0.000 }
gfCNCPoint2[15142] = {X 98.2614, Y 11.2255, Z -3.0000, A 0.000, B 0.000, C 0.000 }
gfCNCPoint2[15143] = {X 98.3697, Y 12.1868, Z -3.0000, A 0.000, B 0.000, C 0.000 }
gfCNCPoint2[15144] = {X 98.3697, Y 12.9781, Z -3.0000, A 0.000, B 0.000, C 0.000 }
gfCNCPoint2[15145] = {X 98.2966, Y 13.7682, Z -3.0000, A 0.000, B 0.000, C 0.000 }
gfCNCPoint2[15146] = {X 98.0804, Y 14.5317, Z -3.0000, A 0.000, B 0.000, C 0.000 }
gfCNCPoint2[15147] = {X 97.7281, Y 15.2426, Z -3.0000, A 0.000, B 0.000, C 0.000 }
gfCNCPoint2[15148] = {X 101.8779, Y 25.5300, Z -3.0000, A 0.000, B 0.000, C 0.000 }
gfCNCPoint2[15149] = {X 106.0167, Y 15.2218, Z -3.0000, A 0.000, B 0.000, C 0.000 }
gfCNCPoint2[15150] = {X 105.6762, Y 14.5288, Z -3.0000, A 0.000, B 0.000, C 0.000 }
gfCNCPoint2[15151] = {X 105.4646, Y 13.7863, Z -3.0000, A 0.000, B 0.000, C 0.000 }
gfCNCPoint2[15152] = {X 105.3885, Y 13.0179, Z -3.0000, A 0.000, B 0.000, C 0.000 }
gfCNCPoint2[15153] = {X 105.3883, Y 12.1868, Z -3.0000, A 0.000, B 0.000, C 0.000 }
gfCNCPoint2[15154] = {X 105.4966, Y 11.2255, Z -3.0000, A 0.000, B 0.000, C 0.000 }
gfCNCPoint2[15155] = {X 105.8161, Y 10.3124, Z -3.0000, A 0.000, B 0.000, C 0.000 }
gfCNCPoint2[15156] = {X 106.3308, Y 9.4933, Z -3.0000, A 0.000, B 0.000, C 0.000 }
gfCNCPoint2[15157] = {X 107.0148, Y 8.8093, Z -3.0000, A 0.000, B 0.000, C 0.000 }
gfCNCPoint2[15158] = {X 107.8339, Y 8.2946, Z -3.0000, A 0.000, B 0.000, C 0.000 }
gfCNCPoint2[15159] = {X 108.7470, Y 7.9751, Z -3.0000, A 0.000, B 0.000, C 0.000 }
gfCNCPoint2[15160] = {X 109.7083, Y 7.8668, Z -3.0000, A 0.000, B 0.000, C 0.000 }
gfCNCPoint2[15161] = {X 117.7916, Y 7.8668, Z -3.0000, A 0.000, B 0.000, C 0.000 }
gfCNCPoint2[15162] = {X 118.7529, Y 7.9751, Z -3.0000, A 0.000, B 0.000, C 0.000 }
gfCNCPoint2[15163] = {X 119.6660, Y 8.2946, Z -3.0000, A 0.000, B 0.000, C 0.000 }
gfCNCPoint2[15164] = {X 120.4851, Y 8.8093, Z -3.0000, A 0.000, B 0.000, C 0.000 }
gfCNCPoint2[15165] = {X 121.1691, Y 9.4933, Z -3.0000, A 0.000, B 0.000, C 0.000 }
gfCNCPoint2[15166] = {X 121.6838, Y 10.3124, Z -3.0000, A 0.000, B 0.000, C 0.000 }
gfCNCPoint2[15167] = {X 122.0033, Y 11.2255, Z -3.0000, A 0.000, B 0.000, C 0.000 }
gfCNCPoint2[15168] = {X 122.1116, Y 12.1868, Z -3.0000, A 0.000, B 0.000, C 0.000 }
gfCNCPoint2[15169] = {X 122.1116, Y 12.9781, Z -3.0000, A 0.000, B 0.000, C 0.000 }
gfCNCPoint2[15170] = {X 122.0103, Y 13.9079, Z -3.0000, A 0.000, B 0.000, C 0.000 }
gfCNCPoint2[15171] = {X 121.7113, Y 14.7941, Z -3.0000, A 0.000, B 0.000, C 0.000 }
gfCNCPoint2[15172] = {X 121.2285, Y 15.5952, Z -3.0000, A 0.000, B 0.000, C 0.000 }
gfCNCPoint2[15173] = {X 120.5847, Y 16.2736, Z -3.0000, A 0.000, B 0.000, C 0.000 }
gfCNCPoint2[15174] = {X 120.5834, Y 40.9139, Z -3.0000, A 0.000, B 0.000, C 0.000 }
gfCNCPoint2[15175] = {X 120.6219, Y 40.9451, Z -3.0000, A 0.000, B 0.000, C 0.000 }
gfCNCPoint2[15176] = {X 121.2454, Y 41.6139, Z -3.0000, A 0.000, B 0.000, C 0.000 }
gfCNCPoint2[15177] = {X 121.7142, Y 42.3989, Z -3.0000, A 0.000, B 0.000, C 0.000 }
gfCNCPoint2[15178] = {X 122.0072, Y 43.2650, Z -3.0000, A 0.000, B 0.000, C 0.000 }
gfCNCPoint2[15179] = {X 122.1114, Y 44.1734, Z -3.0000, A 0.000, B 0.000, C 0.000 }
gfCNCPoint2[15180] = {X 122.1116, Y 45.0000, Z -3.0000, A 0.000, B 0.000, C 0.000 }
gfCNCPoint2[15181] = {X 122.0033, Y 45.9613, Z -3.0000, A 0.000, B 0.000, C 0.000 }
gfCNCPoint2[15182] = {X 121.6838, Y 46.8744, Z -3.0000, A 0.000, B 0.000, C 0.000 }
gfCNCPoint2[15183] = {X 121.1691, Y 47.6935, Z -3.0000, A 0.000, B 0.000, C 0.000 }
gfCNCPoint2[15184] = {X 120.4851, Y 48.3775, Z -3.0000, A 0.000, B 0.000, C 0.000 }
gfCNCPoint2[15185] = {X 119.6660, Y 48.8922, Z -3.0000, A 0.000, B 0.000, C 0.000 }
gfCNCPoint2[15186] = {X 118.7529, Y 49.2117, Z -3.0000, A 0.000, B 0.000, C 0.000 }
gfCNCPoint2[15187] = {X 117.7916, Y 49.3200, Z -3.0000, A 0.000, B 0.000, C 0.000 }
gfCNCPoint2[15188] = {X 111.9185, Y 49.3200, Z -3.0000, A 0.000, B 0.000, C 0.000 }
gfCNCPoint2[15189] = {X 110.9619, Y 49.2128, Z -3.0000, A 0.000, B 0.000, C 0.000 }
gfCNCPoint2[15190] = {X 110.0529, Y 48.8964, Z -3.0000, A 0.000, B 0.000, C 0.000 }
gfCNCPoint2[15191] = {X 109.2365, Y 48.3866, Z -3.0000, A 0.000, B 0.000, C 0.000 }
gfCNCPoint2[15192] = {X 108.5532, Y 47.7087, Z -3.0000, A 0.000, B 0.000, C 0.000 }
gfCNCPoint2[15193] = {X 108.0369, Y 46.8963, Z -3.0000, A 0.000, B 0.000, C 0.000 }
gfCNCPoint2[15194] = {X 107.7134, Y 45.9898, Z -3.0000, A 0.000, B 0.000, C 0.000 }
gfCNCPoint2[15195] = {X 107.5986, Y 45.0341, Z -3.0000, A 0.000, B 0.000, C 0.000 }
gfCNCPoint2[15196] = {X 107.5985, Y 44.1811, Z -3.0000, A 0.000, B 0.000, C 0.000 }
gfCNCPoint2[15197] = {X 107.6344, Y 43.6356, Z -3.0000, A 0.000, B 0.000, C 0.000 }
gfCNCPoint2[15198] = {X 107.7417, Y 43.0994, Z -3.0000, A 0.000, B 0.000, C 0.000 }
gfCNCPoint2[15199] = {X 107.9081, Y 42.6068, Z -3.0000, A 0.000, B 0.000, C 0.000 }
gfCNCPoint2[15200] = {X 108.1348, Y 42.1387, Z -3.0000, A 0.000, B 0.000, C 0.000 }
gfCNCPoint2[15201] = {X 108.5861, Y 41.4658, Z -3.0000, A 0.000, B 0.000, C 0.000 }
gfCNCPoint2[15202] = {X 109.1266, Y 40.8623, Z -3.0000, A 0.000, B 0.000, C 0.000 }
gfCNCPoint2[15203] = {X 109.1265, Y 39.2945, Z -3.0000, A 0.000, B 0.000, C 0.000 }
gfCNCPoint2[15204] = {X 106.1118, Y 46.6615, Z -3.0000, A 0.000, B 0.000, C 0.000 }
gfCNCPoint2[15205] = {X 105.7417, Y 47.3611, Z -3.0000, A 0.000, B 0.000, C 0.000 }
gfCNCPoint2[15206] = {X 105.2502, Y 47.9815, Z -3.0000, A 0.000, B 0.000, C 0.000 }
gfCNCPoint2[15207] = {X 104.6538, Y 48.5018, Z -3.0000, A 0.000, B 0.000, C 0.000 }
gfCNCPoint2[15208] = {X 103.9724, Y 48.9046, Z -3.0000, A 0.000, B 0.000, C 0.000 }
gfCNCPoint2[15209] = {X 103.0287, Y 49.2242, Z -3.0000, A 0.000, B 0.000, C 0.000 }
gfCNCPoint2[15210] = {X 102.0368, Y 49.3191, Z -3.0000, A 0.000, B 0.000, C 0.000 }
gfCNCPoint2[15211] = {X 101.0496, Y 49.1842, Z -3.0000, A 0.000, B 0.000, C 0.000 }
gfCNCPoint2[15212] = {X 100.1195, Y 48.8268, Z -3.0000, A 0.000, B 0.000, C 0.000 }
gfCNCPoint2[15213] = {X 99.2961, Y 48.2657, Z -3.0000, A 0.000, B 0.000, C 0.000 }
gfCNCPoint2[15214] = {X 98.6231, Y 47.5309, Z -3.0000, A 0.000, B 0.000, C 0.000 }
gfCNCPoint2[15215] = {X 98.1363, Y 46.6615, Z -3.0000, A 0.000, B 0.000, C 0.000 }
gfCNCPoint2[15216] = {X 95.1304, Y 39.3101, Z -3.0000, A 0.000, B 0.000, C 0.000 }
gfCNCPoint2[15217] = {X 95.1305, Y 40.9053, Z -3.0000, A 0.000, B 0.000, C 0.000 }
gfCNCPoint2[15218] = {X 95.6595, Y 41.4476, Z -3.0000, A 0.000, B 0.000, C 0.000 }
gfCNCPoint2[15219] = {X 96.0877, Y 42.0725, Z -3.0000, A 0.000, B 0.000, C 0.000 }
gfCNCPoint2[15220] = {X 96.3309, Y 42.5741, Z -3.0000, A 0.000, B 0.000, C 0.000 }
gfCNCPoint2[15221] = {X 96.5088, Y 43.1024, Z -3.0000, A 0.000, B 0.000, C 0.000 }
gfCNCPoint2[15222] = {X 96.6187, Y 43.6496, Z -3.0000, A 0.000, B 0.000, C 0.000 }
gfCNCPoint2[15223] = {X 96.6585, Y 44.2063, Z -3.0000, A 0.000, B 0.000, C 0.000 }
gfCNCPoint2[15224] = {X 96.6583, Y 45.0415, Z -3.0000, A 0.000, B 0.000, C 0.000 }
gfCNCPoint2[15225] = {X 96.5422, Y 45.9960, Z -3.0000, A 0.000, B 0.000, C 0.000 }
gfCNCPoint2[15226] = {X 96.2178, Y 46.9011, Z -3.0000, A 0.000, B 0.000, C 0.000 }
gfCNCPoint2[15227] = {X 95.7012, Y 47.7120, Z -3.0000, A 0.000, B 0.000, C 0.000 }
gfCNCPoint2[15228] = {X 95.0181, Y 48.3886, Z -3.0000, A 0.000, B 0.000, C 0.000 }
gfCNCPoint2[15229] = {X 94.2022, Y 48.8973, Z -3.0000, A 0.000, B 0.000, C 0.000 }
gfCNCPoint2[15230] = {X 93.2940, Y 49.2130, Z -3.0000, A 0.000, B 0.000, C 0.000 }
gfCNCPoint2[15231] = {X 92.3385, Y 49.3200, Z -3.0000, A 0.000, B 0.000, C 0.000 }
gfCNCPoint2[15232] = {X 85.8951, Y 49.3200, Z -3.0000, A 0.000, B 0.000, C 0.000 }
gfCNCPoint2[15233] = {X 84.9387, Y 49.2128, Z -3.0000, A 0.000, B 0.000, C 0.000 }
gfCNCPoint2[15234] = {X 84.0297, Y 48.8965, Z -3.0000, A 0.000, B 0.000, C 0.000 }
gfCNCPoint2[15235] = {X 83.2134, Y 48.3869, Z -3.0000, A 0.000, B 0.000, C 0.000 }
gfCNCPoint2[15236] = {X 82.5301, Y 47.7091, Z -3.0000, A 0.000, B 0.000, C 0.000 }
gfCNCPoint2[15237] = {X 82.0138, Y 46.8970, Z -3.0000, A 0.000, B 0.000, C 0.000 }
gfCNCPoint2[15238] = {X 81.6902, Y 45.9906, Z -3.0000, A 0.000, B 0.000, C 0.000 }
gfCNCPoint2[15239] = {X 81.5752, Y 45.0351, Z -3.0000, A 0.000, B 0.000, C 0.000 }
gfCNCPoint2[15240] = {X 81.5751, Y 44.2069, Z -3.0000, A 0.000, B 0.000, C 0.000 }
gfCNCPoint2[15241] = {X 81.6807, Y 43.2777, Z -3.0000, A 0.000, B 0.000, C 0.000 }
gfCNCPoint2[15242] = {X 81.9812, Y 42.3922, Z -3.0000, A 0.000, B 0.000, C 0.000 }
gfCNCPoint2[15243] = {X 82.4627, Y 41.5905, Z -3.0000, A 0.000, B 0.000, C 0.000 }
gfCNCPoint2[15244] = {X 83.1034, Y 40.9093, Z -3.0000, A 0.000, B 0.000, C 0.000 }
gfCNCPoint2[15245] = {X 83.1033, Y 28.5920, Z -3.0000, A 0.000, B 0.000, C 0.000 }
gfCNCPoint2[15246] = {X 79.1033, Y 28.5920, Z -3.0000, A 0.000, B 0.000, C 0.000 }
gfCNCPoint2[15247] = {X 83.1833, Y 28.5920, Z -3.0000, A 0.000, B 0.000, C 0.000 }
gfCNCPoint2[15248] = {X 83.1831, Y 16.2373, Z -3.0000, A 0.000, B 0.000, C 0.000 }
gfCNCPoint2[15249] = {X 82.5448, Y 15.5767, Z -3.0000, A 0.000, B 0.000, C 0.000 }
gfCNCPoint2[15250] = {X 82.0637, Y 14.7942, Z -3.0000, A 0.000, B 0.000, C 0.000 }
gfCNCPoint2[15251] = {X 81.7625, Y 13.9264, Z -3.0000, A 0.000, B 0.000, C 0.000 }
gfCNCPoint2[15252] = {X 81.6552, Y 13.0142, Z -3.0000, A 0.000, B 0.000, C 0.000 }
gfCNCPoint2[15253] = {X 81.6551, Y 12.1868, Z -3.0000, A 0.000, B 0.000, C 0.000 }
gfCNCPoint2[15254] = {X 81.7614, Y 11.2433, Z -3.0000, A 0.000, B 0.000, C 0.000 }
gfCNCPoint2[15255] = {X 82.0750, Y 10.3472, Z -3.0000, A 0.000, B 0.000, C 0.000 }
gfCNCPoint2[15256] = {X 82.5801, Y 9.5432, Z -3.0000, A 0.000, B 0.000, C 0.000 }
gfCNCPoint2[15257] = {X 83.2515, Y 8.8719, Z -3.0000, A 0.000, B 0.000, C 0.000 }
gfCNCPoint2[15258] = {X 84.0554, Y 8.3667, Z -3.0000, A 0.000, B 0.000, C 0.000 }
gfCNCPoint2[15259] = {X 84.9516, Y 8.0531, Z -3.0000, A 0.000, B 0.000, C 0.000 }
gfCNCPoint2[15260] = {X 85.8951, Y 7.9468, Z -3.0000, A 0.000, B 0.000, C 0.000 }
gfCNCPoint2[15261] = {X 94.0497, Y 7.9468, Z -3.0000, A 0.000, B 0.000, C 0.000 }
gfCNCPoint2[15262] = {X 94.9932, Y 8.0531, Z -3.0000, A 0.000, B 0.000, C 0.000 }
gfCNCPoint2[15263] = {X 95.8893, Y 8.3667, Z -3.0000, A 0.000, B 0.000, C 0.000 }
gfCNCPoint2[15264] = {X 96.6933, Y 8.8718, Z -3.0000, A 0.000, B 0.000, C 0.000 }
gfCNCPoint2[15265] = {X 97.3646, Y 9.5432, Z -3.0000, A 0.000, B 0.000, C 0.000 }
gfCNCPoint2[15266] = {X 97.8698, Y 10.3471, Z -3.0000, A 0.000, B 0.000, C 0.000 }
gfCNCPoint2[15267] = {X 98.1834, Y 11.2433, Z -3.0000, A 0.000, B 0.000, C 0.000 }
gfCNCPoint2[15268] = {X 98.2897, Y 12.1868, Z -3.0000, A 0.000, B 0.000, C 0.000 }
gfCNCPoint2[15269] = {X 98.2897, Y 12.9781, Z -3.0000, A 0.000, B 0.000, C 0.000 }
gfCNCPoint2[15270] = {X 98.2155, Y 13.7668, Z -3.0000, A 0.000, B 0.000, C 0.000 }
gfCNCPoint2[15271] = {X 97.9960, Y 14.5279, Z -3.0000, A 0.000, B 0.000, C 0.000 }
gfCNCPoint2[15272] = {X 97.6387, Y 15.2348, Z -3.0000, A 0.000, B 0.000, C 0.000 }
gfCNCPoint2[15273] = {X 101.8779, Y 25.7436, Z -3.0000, A 0.000, B 0.000, C 0.000 }
gfCNCPoint2[15274] = {X 101.9522, Y 25.5598, Z -3.0000, A 0.000, B 0.000, C 0.000 }
gfCNCPoint2[15275] = {X 106.1059, Y 15.2143, Z -3.0000, A 0.000, B 0.000, C 0.000 }
gfCNCPoint2[15276] = {X 105.7605, Y 14.5249, Z -3.0000, A 0.000, B 0.000, C 0.000 }
gfCNCPoint2[15277] = {X 105.5457, Y 13.7844, Z -3.0000, A 0.000, B 0.000, C 0.000 }
gfCNCPoint2[15278] = {X 105.4685, Y 13.0172, Z -3.0000, A 0.000, B 0.000, C 0.000 }
gfCNCPoint2[15279] = {X 105.4683, Y 12.1868, Z -3.0000, A 0.000, B 0.000, C 0.000 }
gfCNCPoint2[15280] = {X 105.5746, Y 11.2433, Z -3.0000, A 0.000, B 0.000, C 0.000 }
gfCNCPoint2[15281] = {X 105.8882, Y 10.3471, Z -3.0000, A 0.000, B 0.000, C 0.000 }
gfCNCPoint2[15282] = {X 106.3933, Y 9.5432, Z -3.0000, A 0.000, B 0.000, C 0.000 }
gfCNCPoint2[15283] = {X 107.0647, Y 8.8718, Z -3.0000, A 0.000, B 0.000, C 0.000 }
gfCNCPoint2[15284] = {X 107.8686, Y 8.3667, Z -3.0000, A 0.000, B 0.000, C 0.000 }
gfCNCPoint2[15285] = {X 108.7648, Y 8.0531, Z -3.0000, A 0.000, B 0.000, C 0.000 }
gfCNCPoint2[15286] = {X 109.7083, Y 7.9468, Z -3.0000, A 0.000, B 0.000, C 0.000 }
gfCNCPoint2[15287] = {X 117.7916, Y 7.9468, Z -3.0000, A 0.000, B 0.000, C 0.000 }
gfCNCPoint2[15288] = {X 118.7351, Y 8.0531, Z -3.0000, A 0.000, B 0.000, C 0.000 }
gfCNCPoint2[15289] = {X 119.6312, Y 8.3667, Z -3.0000, A 0.000, B 0.000, C 0.000 }
gfCNCPoint2[15290] = {X 120.4352, Y 8.8718, Z -3.0000, A 0.000, B 0.000, C 0.000 }
gfCNCPoint2[15291] = {X 121.1065, Y 9.5432, Z -3.0000, A 0.000, B 0.000, C 0.000 }
gfCNCPoint2[15292] = {X 121.6117, Y 10.3471, Z -3.0000, A 0.000, B 0.000, C 0.000 }
gfCNCPoint2[15293] = {X 121.9253, Y 11.2433, Z -3.0000, A 0.000, B 0.000, C 0.000 }
gfCNCPoint2[15294] = {X 122.0316, Y 12.1868, Z -3.0000, A 0.000, B 0.000, C 0.000 }
gfCNCPoint2[15295] = {X 122.0316, Y 12.9781, Z -3.0000, A 0.000, B 0.000, C 0.000 }
gfCNCPoint2[15296] = {X 121.9302, Y 13.8997, Z -3.0000, A 0.000, B 0.000, C 0.000 }
gfCNCPoint2[15297] = {X 121.6309, Y 14.7772, Z -3.0000, A 0.000, B 0.000, C 0.000 }
gfCNCPoint2[15298] = {X 121.1480, Y 15.5687, Z -3.0000, A 0.000, B 0.000, C 0.000 }
gfCNCPoint2[15299] = {X 120.5047, Y 16.2363, Z -3.0000, A 0.000, B 0.000, C 0.000 }
gfCNCPoint2[15300] = {X 120.5034, Y 40.9519, Z -3.0000, A 0.000, B 0.000, C 0.000 }
gfCNCPoint2[15301] = {X 120.5704, Y 41.0063, Z -3.0000, A 0.000, B 0.000, C 0.000 }
gfCNCPoint2[15302] = {X 121.1820, Y 41.6627, Z -3.0000, A 0.000, B 0.000, C 0.000 }
gfCNCPoint2[15303] = {X 121.6418, Y 42.4330, Z -3.0000, A 0.000, B 0.000, C 0.000 }
gfCNCPoint2[15304] = {X 121.9292, Y 43.2828, Z -3.0000, A 0.000, B 0.000, C 0.000 }
gfCNCPoint2[15305] = {X 122.0314, Y 44.1740, Z -3.0000, A 0.000, B 0.000, C 0.000 }
gfCNCPoint2[15306] = {X 122.0316, Y 45.0000, Z -3.0000, A 0.000, B 0.000, C 0.000 }
gfCNCPoint2[15307] = {X 121.9253, Y 45.9435, Z -3.0000, A 0.000, B 0.000, C 0.000 }
gfCNCPoint2[15308] = {X 121.6117, Y 46.8397, Z -3.0000, A 0.000, B 0.000, C 0.000 }
gfCNCPoint2[15309] = {X 121.1065, Y 47.6436, Z -3.0000, A 0.000, B 0.000, C 0.000 }
gfCNCPoint2[15310] = {X 120.4352, Y 48.3150, Z -3.0000, A 0.000, B 0.000, C 0.000 }
gfCNCPoint2[15311] = {X 119.6312, Y 48.8201, Z -3.0000, A 0.000, B 0.000, C 0.000 }
gfCNCPoint2[15312] = {X 118.7351, Y 49.1337, Z -3.0000, A 0.000, B 0.000, C 0.000 }
gfCNCPoint2[15313] = {X 117.7916, Y 49.2400, Z -3.0000, A 0.000, B 0.000, C 0.000 }
gfCNCPoint2[15314] = {X 111.9185, Y 49.2400, Z -3.0000, A 0.000, B 0.000, C 0.000 }
gfCNCPoint2[15315] = {X 110.9797, Y 49.1348, Z -3.0000, A 0.000, B 0.000, C 0.000 }
gfCNCPoint2[15316] = {X 110.0874, Y 48.8242, Z -3.0000, A 0.000, B 0.000, C 0.000 }
gfCNCPoint2[15317] = {X 109.2861, Y 48.3239, Z -3.0000, A 0.000, B 0.000, C 0.000 }
gfCNCPoint2[15318] = {X 108.6155, Y 47.6585, Z -3.0000, A 0.000, B 0.000, C 0.000 }
gfCNCPoint2[15319] = {X 108.1088, Y 46.8612, Z -3.0000, A 0.000, B 0.000, C 0.000 }
gfCNCPoint2[15320] = {X 107.7913, Y 45.9714, Z -3.0000, A 0.000, B 0.000, C 0.000 }
gfCNCPoint2[15321] = {X 107.6786, Y 45.0335, Z -3.0000, A 0.000, B 0.000, C 0.000 }
gfCNCPoint2[15322] = {X 107.6785, Y 44.1811, Z -3.0000, A 0.000, B 0.000, C 0.000 }
gfCNCPoint2[15323] = {X 107.7137, Y 43.6461, Z -3.0000, A 0.000, B 0.000, C 0.000 }
gfCNCPoint2[15324] = {X 107.8189, Y 43.1203, Z -3.0000, A 0.000, B 0.000, C 0.000 }
gfCNCPoint2[15325] = {X 107.9822, Y 42.6371, Z -3.0000, A 0.000, B 0.000, C 0.000 }
gfCNCPoint2[15326] = {X 108.2045, Y 42.1780, Z -3.0000, A 0.000, B 0.000, C 0.000 }
gfCNCPoint2[15327] = {X 108.6598, Y 41.5014, Z -3.0000, A 0.000, B 0.000, C 0.000 }
gfCNCPoint2[15328] = {X 109.2066, Y 40.8962, Z -3.0000, A 0.000, B 0.000, C 0.000 }
gfCNCPoint2[15329] = {X 109.2065, Y 39.1629, Z -3.0000, A 0.000, B 0.000, C 0.000 }
gfCNCPoint2[15330] = {X 109.0939, Y 39.1629, Z -3.0000, A 0.000, B 0.000, C 0.000 }
gfCNCPoint2[15331] = {X 106.0379, Y 46.6307, Z -3.0000, A 0.000, B 0.000, C 0.000 }
gfCNCPoint2[15332] = {X 105.6747, Y 47.3174, Z -3.0000, A 0.000, B 0.000, C 0.000 }
gfCNCPoint2[15333] = {X 105.1923, Y 47.9263, Z -3.0000, A 0.000, B 0.000, C 0.000 }
gfCNCPoint2[15334] = {X 104.6069, Y 48.4370, Z -3.0000, A 0.000, B 0.000, C 0.000 }
gfCNCPoint2[15335] = {X 103.9382, Y 48.8323, Z -3.0000, A 0.000, B 0.000, C 0.000 }
gfCNCPoint2[15336] = {X 103.0119, Y 49.1460, Z -3.0000, A 0.000, B 0.000, C 0.000 }
gfCNCPoint2[15337] = {X 102.0384, Y 49.2391, Z -3.0000, A 0.000, B 0.000, C 0.000 }
gfCNCPoint2[15338] = {X 101.0695, Y 49.1068, Z -3.0000, A 0.000, B 0.000, C 0.000 }
gfCNCPoint2[15339] = {X 100.1566, Y 48.7559, Z -3.0000, A 0.000, B 0.000, C 0.000 }
gfCNCPoint2[15340] = {X 99.3484, Y 48.2052, Z -3.0000, A 0.000, B 0.000, C 0.000 }
gfCNCPoint2[15341] = {X 98.6879, Y 47.4840, Z -3.0000, A 0.000, B 0.000, C 0.000 }
gfCNCPoint2[15342] = {X 98.2102, Y 46.6307, Z -3.0000, A 0.000, B 0.000, C 0.000 }
gfCNCPoint2[15343] = {X 95.0504, Y 38.9030, Z -3.0000, A 0.000, B 0.000, C 0.000 }
gfCNCPoint2[15344] = {X 95.0505, Y 40.9422, Z -3.0000, A 0.000, B 0.000, C 0.000 }
gfCNCPoint2[15345] = {X 95.5860, Y 41.4843, Z -3.0000, A 0.000, B 0.000, C 0.000 }
gfCNCPoint2[15346] = {X 96.0181, Y 42.1119, Z -3.0000, A 0.000, B 0.000, C 0.000 }
gfCNCPoint2[15347] = {X 96.2569, Y 42.6044, Z -3.0000, A 0.000, B 0.000, C 0.000 }
gfCNCPoint2[15348] = {X 96.4315, Y 43.1231, Z -3.0000, A 0.000, B 0.000, C 0.000 }
gfCNCPoint2[15349] = {X 96.5394, Y 43.6604, Z -3.0000, A 0.000, B 0.000, C 0.000 }
gfCNCPoint2[15350] = {X 96.5785, Y 44.2070, Z -3.0000, A 0.000, B 0.000, C 0.000 }
gfCNCPoint2[15351] = {X 96.5783, Y 45.0408, Z -3.0000, A 0.000, B 0.000, C 0.000 }
gfCNCPoint2[15352] = {X 96.4643, Y 45.9775, Z -3.0000, A 0.000, B 0.000, C 0.000 }
gfCNCPoint2[15353] = {X 96.1459, Y 46.8659, Z -3.0000, A 0.000, B 0.000, C 0.000 }
gfCNCPoint2[15354] = {X 95.6389, Y 47.6618, Z -3.0000, A 0.000, B 0.000, C 0.000 }
gfCNCPoint2[15355] = {X 94.9685, Y 48.3258, Z -3.0000, A 0.000, B 0.000, C 0.000 }
gfCNCPoint2[15356] = {X 94.1677, Y 48.8251, Z -3.0000, A 0.000, B 0.000, C 0.000 }
gfCNCPoint2[15357] = {X 93.2764, Y 49.1350, Z -3.0000, A 0.000, B 0.000, C 0.000 }
gfCNCPoint2[15358] = {X 92.3385, Y 49.2400, Z -3.0000, A 0.000, B 0.000, C 0.000 }
gfCNCPoint2[15359] = {X 85.8951, Y 49.2400, Z -3.0000, A 0.000, B 0.000, C 0.000 }
gfCNCPoint2[15360] = {X 84.9564, Y 49.1348, Z -3.0000, A 0.000, B 0.000, C 0.000 }
gfCNCPoint2[15361] = {X 84.0643, Y 48.8244, Z -3.0000, A 0.000, B 0.000, C 0.000 }
gfCNCPoint2[15362] = {X 83.2631, Y 48.3242, Z -3.0000, A 0.000, B 0.000, C 0.000 }
gfCNCPoint2[15363] = {X 82.5924, Y 47.6590, Z -3.0000, A 0.000, B 0.000, C 0.000 }
gfCNCPoint2[15364] = {X 82.0857, Y 46.8618, Z -3.0000, A 0.000, B 0.000, C 0.000 }
gfCNCPoint2[15365] = {X 81.7681, Y 45.9723, Z -3.0000, A 0.000, B 0.000, C 0.000 }
gfCNCPoint2[15366] = {X 81.6552, Y 45.0345, Z -3.0000, A 0.000, B 0.000, C 0.000 }
gfCNCPoint2[15367] = {X 81.6551, Y 44.2074, Z -3.0000, A 0.000, B 0.000, C 0.000 }
gfCNCPoint2[15368] = {X 81.7608, Y 43.2863, Z -3.0000, A 0.000, B 0.000, C 0.000 }
gfCNCPoint2[15369] = {X 82.0615, Y 42.4092, Z -3.0000, A 0.000, B 0.000, C 0.000 }
gfCNCPoint2[15370] = {X 82.5431, Y 41.6169, Z -3.0000, A 0.000, B 0.000, C 0.000 }
gfCNCPoint2[15371] = {X 83.1834, Y 40.9463, Z -3.0000, A 0.000, B 0.000, C 0.000 }
gfCNCPoint2[15372] = {X 83.1833, Y 28.5920, Z -3.0000, A 0.000, B 0.000, C 0.000 }
gfCNCPoint2[15373] = {X 79.1833, Y 28.5920, Z -3.0000, A 0.000, B 0.000, C 0.000 }
gfCNCPoint2[15374] = {X 83.2633, Y 28.5920, Z -3.0000, A 0.000, B 0.000, C 0.000 }
gfCNCPoint2[15375] = {X 83.2631, Y 16.1996, Z -3.0000, A 0.000, B 0.000, C 0.000 }
gfCNCPoint2[15376] = {X 82.6253, Y 15.5498, Z -3.0000, A 0.000, B 0.000, C 0.000 }
gfCNCPoint2[15377] = {X 82.1441, Y 14.7768, Z -3.0000, A 0.000, B 0.000, C 0.000 }
gfCNCPoint2[15378] = {X 81.8426, Y 13.9176, Z -3.0000, A 0.000, B 0.000, C 0.000 }
gfCNCPoint2[15379] = {X 81.7352, Y 13.0135, Z -3.0000, A 0.000, B 0.000, C 0.000 }
gfCNCPoint2[15380] = {X 81.7351, Y 12.1868, Z -3.0000, A 0.000, B 0.000, C 0.000 }
gfCNCPoint2[15381] = {X 81.8394, Y 11.2611, Z -3.0000, A 0.000, B 0.000, C 0.000 }
gfCNCPoint2[15382] = {X 82.1470, Y 10.3819, Z -3.0000, A 0.000, B 0.000, C 0.000 }
gfCNCPoint2[15383] = {X 82.6427, Y 9.5931, Z -3.0000, A 0.000, B 0.000, C 0.000 }
gfCNCPoint2[15384] = {X 83.3014, Y 8.9344, Z -3.0000, A 0.000, B 0.000, C 0.000 }
gfCNCPoint2[15385] = {X 84.0901, Y 8.4388, Z -3.0000, A 0.000, B 0.000, C 0.000 }
gfCNCPoint2[15386] = {X 84.9694, Y 8.1311, Z -3.0000, A 0.000, B 0.000, C 0.000 }
gfCNCPoint2[15387] = {X 85.8951, Y 8.0268, Z -3.0000, A 0.000, B 0.000, C 0.000 }
gfCNCPoint2[15388] = {X 94.0497, Y 8.0268, Z -3.0000, A 0.000, B 0.000, C 0.000 }
gfCNCPoint2[15389] = {X 94.9754, Y 8.1311, Z -3.0000, A 0.000, B 0.000, C 0.000 }
gfCNCPoint2[15390] = {X 95.8546, Y 8.4388, Z -3.0000, A 0.000, B 0.000, C 0.000 }
gfCNCPoint2[15391] = {X 96.6434, Y 8.9344, Z -3.0000, A 0.000, B 0.000, C 0.000 }
gfCNCPoint2[15392] = {X 97.3021, Y 9.5931, Z -3.0000, A 0.000, B 0.000, C 0.000 }
gfCNCPoint2[15393] = {X 97.7977, Y 10.3819, Z -3.0000, A 0.000, B 0.000, C 0.000 }
gfCNCPoint2[15394] = {X 98.1054, Y 11.2611, Z -3.0000, A 0.000, B 0.000, C 0.000 }
gfCNCPoint2[15395] = {X 98.2097, Y 12.1868, Z -3.0000, A 0.000, B 0.000, C 0.000 }
gfCNCPoint2[15396] = {X 98.2097, Y 12.9781, Z -3.0000, A 0.000, B 0.000, C 0.000 }
gfCNCPoint2[15397] = {X 98.1343, Y 13.7661, Z -3.0000, A 0.000, B 0.000, C 0.000 }
gfCNCPoint2[15398] = {X 97.9111, Y 14.5256, Z -3.0000, A 0.000, B 0.000, C 0.000 }
gfCNCPoint2[15399] = {X 97.5480, Y 15.2290, Z -3.0000, A 0.000, B 0.000, C 0.000 }
gfCNCPoint2[15400] = {X 101.8773, Y 25.9562, Z -3.0000, A 0.000, B 0.000, C 0.000 }
gfCNCPoint2[15401] = {X 101.9785, Y 25.7088, Z -3.0000, A 0.000, B 0.000, C 0.000 }
gfCNCPoint2[15402] = {X 106.1954, Y 15.2063, Z -3.0000, A 0.000, B 0.000, C 0.000 }
gfCNCPoint2[15403] = {X 105.8449, Y 14.5207, Z -3.0000, A 0.000, B 0.000, C 0.000 }
gfCNCPoint2[15404] = {X 105.6268, Y 13.7823, Z -3.0000, A 0.000, B 0.000, C 0.000 }
gfCNCPoint2[15405] = {X 105.5485, Y 13.0164, Z -3.0000, A 0.000, B 0.000, C 0.000 }
gfCNCPoint2[15406] = {X 105.5483, Y 12.1868, Z -3.0000, A 0.000, B 0.000, C 0.000 }
gfCNCPoint2[15407] = {X 105.6526, Y 11.2611, Z -3.0000, A 0.000, B 0.000, C 0.000 }
gfCNCPoint2[15408] = {X 105.9602, Y 10.3819, Z -3.0000, A 0.000, B 0.000, C 0.000 }
gfCNCPoint2[15409] = {X 106.4559, Y 9.5931, Z -3.0000, A 0.000, B 0.000, C 0.000 }
gfCNCPoint2[15410] = {X 107.1146, Y 8.9344, Z -3.0000, A 0.000, B 0.000, C 0.000 }
gfCNCPoint2[15411] = {X 107.9033, Y 8.4388, Z -3.0000, A 0.000, B 0.000, C 0.000 }
gfCNCPoint2[15412] = {X 108.7826, Y 8.1311, Z -3.0000, A 0.000, B 0.000, C 0.000 }
gfCNCPoint2[15413] = {X 109.7083, Y 8.0268, Z -3.0000, A 0.000, B 0.000, C 0.000 }
gfCNCPoint2[15414] = {X 117.7916, Y 8.0268, Z -3.0000, A 0.000, B 0.000, C 0.000 }
gfCNCPoint2[15415] = {X 118.7173, Y 8.1311, Z -3.0000, A 0.000, B 0.000, C 0.000 }
gfCNCPoint2[15416] = {X 119.5965, Y 8.4388, Z -3.0000, A 0.000, B 0.000, C 0.000 }
gfCNCPoint2[15417] = {X 120.3853, Y 8.9344, Z -3.0000, A 0.000, B 0.000, C 0.000 }
gfCNCPoint2[15418] = {X 121.0440, Y 9.5931, Z -3.0000, A 0.000, B 0.000, C 0.000 }
gfCNCPoint2[15419] = {X 121.5396, Y 10.3819, Z -3.0000, A 0.000, B 0.000, C 0.000 }
gfCNCPoint2[15420] = {X 121.8473, Y 11.2611, Z -3.0000, A 0.000, B 0.000, C 0.000 }
gfCNCPoint2[15421] = {X 121.9516, Y 12.1868, Z -3.0000, A 0.000, B 0.000, C 0.000 }
gfCNCPoint2[15422] = {X 121.9516, Y 12.9781, Z -3.0000, A 0.000, B 0.000, C 0.000 }
gfCNCPoint2[15423] = {X 121.8501, Y 13.8915, Z -3.0000, A 0.000, B 0.000, C 0.000 }
gfCNCPoint2[15424] = {X 121.5505, Y 14.7602, Z -3.0000, A 0.000, B 0.000, C 0.000 }
gfCNCPoint2[15425] = {X 121.0675, Y 15.5420, Z -3.0000, A 0.000, B 0.000, C 0.000 }
gfCNCPoint2[15426] = {X 120.4247, Y 16.1986, Z -3.0000, A 0.000, B 0.000, C 0.000 }
gfCNCPoint2[15427] = {X 120.4234, Y 40.9900, Z -3.0000, A 0.000, B 0.000, C 0.000 }
gfCNCPoint2[15428] = {X 120.5190, Y 41.0676, Z -3.0000, A 0.000, B 0.000, C 0.000 }
gfCNCPoint2[15429] = {X 121.1186, Y 41.7115, Z -3.0000, A 0.000, B 0.000, C 0.000 }
gfCNCPoint2[15430] = {X 121.5694, Y 42.4671, Z -3.0000, A 0.000, B 0.000, C 0.000 }
gfCNCPoint2[15431] = {X 121.8512, Y 43.3006, Z -3.0000, A 0.000, B 0.000, C 0.000 }
gfCNCPoint2[15432] = {X 121.9514, Y 44.1747, Z -3.0000, A 0.000, B 0.000, C 0.000 }
gfCNCPoint2[15433] = {X 121.9516, Y 45.0000, Z -3.0000, A 0.000, B 0.000, C 0.000 }
gfCNCPoint2[15434] = {X 121.8473, Y 45.9257, Z -3.0000, A 0.000, B 0.000, C 0.000 }
gfCNCPoint2[15435] = {X 121.5396, Y 46.8050, Z -3.0000, A 0.000, B 0.000, C 0.000 }
gfCNCPoint2[15436] = {X 121.0440, Y 47.5937, Z -3.0000, A 0.000, B 0.000, C 0.000 }
gfCNCPoint2[15437] = {X 120.3853, Y 48.2524, Z -3.0000, A 0.000, B 0.000, C 0.000 }
gfCNCPoint2[15438] = {X 119.5965, Y 48.7480, Z -3.0000, A 0.000, B 0.000, C 0.000 }
gfCNCPoint2[15439] = {X 118.7173, Y 49.0557, Z -3.0000, A 0.000, B 0.000, C 0.000 }
gfCNCPoint2[15440] = {X 117.7916, Y 49.1600, Z -3.0000, A 0.000, B 0.000, C 0.000 }
gfCNCPoint2[15441] = {X 111.9185, Y 49.1600, Z -3.0000, A 0.000, B 0.000, C 0.000 }
gfCNCPoint2[15442] = {X 110.9974, Y 49.0567, Z -3.0000, A 0.000, B 0.000, C 0.000 }
gfCNCPoint2[15443] = {X 110.1220, Y 48.7521, Z -3.0000, A 0.000, B 0.000, C 0.000 }
gfCNCPoint2[15444] = {X 109.3358, Y 48.2612, Z -3.0000, A 0.000, B 0.000, C 0.000 }
gfCNCPoint2[15445] = {X 108.6778, Y 47.6084, Z -3.0000, A 0.000, B 0.000, C 0.000 }
gfCNCPoint2[15446] = {X 108.1807, Y 46.8261, Z -3.0000, A 0.000, B 0.000, C 0.000 }
gfCNCPoint2[15447] = {X 107.8691, Y 45.9531, Z -3.0000, A 0.000, B 0.000, C 0.000 }
gfCNCPoint2[15448] = {X 107.7586, Y 45.0328, Z -3.0000, A 0.000, B 0.000, C 0.000 }
gfCNCPoint2[15449] = {X 107.7585, Y 44.1811, Z -3.0000, A 0.000, B 0.000, C 0.000 }
gfCNCPoint2[15450] = {X 107.7931, Y 43.6566, Z -3.0000, A 0.000, B 0.000, C 0.000 }
gfCNCPoint2[15451] = {X 107.8962, Y 43.1411, Z -3.0000, A 0.000, B 0.000, C 0.000 }
gfCNCPoint2[15452] = {X 108.0562, Y 42.6674, Z -3.0000, A 0.000, B 0.000, C 0.000 }
gfCNCPoint2[15453] = {X 108.2742, Y 42.2173, Z -3.0000, A 0.000, B 0.000, C 0.000 }
gfCNCPoint2[15454] = {X 108.7335, Y 41.5370, Z -3.0000, A 0.000, B 0.000, C 0.000 }
gfCNCPoint2[15455] = {X 109.2866, Y 40.9305, Z -3.0000, A 0.000, B 0.000, C 0.000 }
gfCNCPoint2[15456] = {X 109.2865, Y 39.0829, Z -3.0000, A 0.000, B 0.000, C 0.000 }
gfCNCPoint2[15457] = {X 109.0402, Y 39.0829, Z -3.0000, A 0.000, B 0.000, C 0.000 }
gfCNCPoint2[15458] = {X 105.9641, Y 46.5999, Z -3.0000, A 0.000, B 0.000, C 0.000 }
gfCNCPoint2[15459] = {X 105.6077, Y 47.2737, Z -3.0000, A 0.000, B 0.000, C 0.000 }
gfCNCPoint2[15460] = {X 105.1344, Y 47.8711, Z -3.0000, A 0.000, B 0.000, C 0.000 }
gfCNCPoint2[15461] = {X 104.5601, Y 48.3721, Z -3.0000, A 0.000, B 0.000, C 0.000 }
gfCNCPoint2[15462] = {X 103.9040, Y 48.7600, Z -3.0000, A 0.000, B 0.000, C 0.000 }
gfCNCPoint2[15463] = {X 102.9952, Y 49.0678, Z -3.0000, A 0.000, B 0.000, C 0.000 }
gfCNCPoint2[15464] = {X 102.0400, Y 49.1592, Z -3.0000, A 0.000, B 0.000, C 0.000 }
gfCNCPoint2[15465] = {X 101.0894, Y 49.0293, Z -3.0000, A 0.000, B 0.000, C 0.000 }
gfCNCPoint2[15466] = {X 100.1937, Y 48.6850, Z -3.0000, A 0.000, B 0.000, C 0.000 }
gfCNCPoint2[15467] = {X 99.4008, Y 48.1448, Z -3.0000, A 0.000, B 0.000, C 0.000 }
gfCNCPoint2[15468] = {X 98.7527, Y 47.4372, Z -3.0000, A 0.000, B 0.000, C 0.000 }
gfCNCPoint2[15469] = {X 98.2840, Y 46.5999, Z -3.0000, A 0.000, B 0.000, C 0.000 }
gfCNCPoint2[15470] = {X 94.9703, Y 38.4959, Z -3.0000, A 0.000, B 0.000, C 0.000 }
gfCNCPoint2[15471] = {X 94.9705, Y 40.9795, Z -3.0000, A 0.000, B 0.000, C 0.000 }
gfCNCPoint2[15472] = {X 95.5126, Y 41.5211, Z -3.0000, A 0.000, B 0.000, C 0.000 }
gfCNCPoint2[15473] = {X 95.9485, Y 42.1513, Z -3.0000, A 0.000, B 0.000, C 0.000 }
gfCNCPoint2[15474] = {X 96.1828, Y 42.6347, Z -3.0000, A 0.000, B 0.000, C 0.000 }
gfCNCPoint2[15475] = {X 96.3543, Y 43.1438, Z -3.0000, A 0.000, B 0.000, C 0.000 }
gfCNCPoint2[15476] = {X 96.4602, Y 43.6711, Z -3.0000, A 0.000, B 0.000, C 0.000 }
gfCNCPoint2[15477] = {X 96.4985, Y 44.2076, Z -3.0000, A 0.000, B 0.000, C 0.000 }
gfCNCPoint2[15478] = {X 96.4983, Y 45.0400, Z -3.0000, A 0.000, B 0.000, C 0.000 }
gfCNCPoint2[15479] = {X 96.3865, Y 45.9591, Z -3.0000, A 0.000, B 0.000, C 0.000 }
gfCNCPoint2[15480] = {X 96.0741, Y 46.8306, Z -3.0000, A 0.000, B 0.000, C 0.000 }
gfCNCPoint2[15481] = {X 95.5767, Y 47.6115, Z -3.0000, A 0.000, B 0.000, C 0.000 }
gfCNCPoint2[15482] = {X 94.9188, Y 48.2631, Z -3.0000, A 0.000, B 0.000, C 0.000 }
gfCNCPoint2[15483] = {X 94.1332, Y 48.7530, Z -3.0000, A 0.000, B 0.000, C 0.000 }
gfCNCPoint2[15484] = {X 93.2587, Y 49.0570, Z -3.0000, A 0.000, B 0.000, C 0.000 }
gfCNCPoint2[15485] = {X 92.3385, Y 49.1600, Z -3.0000, A 0.000, B 0.000, C 0.000 }
gfCNCPoint2[15486] = {X 85.8951, Y 49.1600, Z -3.0000, A 0.000, B 0.000, C 0.000 }
gfCNCPoint2[15487] = {X 84.9741, Y 49.0568, Z -3.0000, A 0.000, B 0.000, C 0.000 }
gfCNCPoint2[15488] = {X 84.0988, Y 48.7522, Z -3.0000, A 0.000, B 0.000, C 0.000 }
gfCNCPoint2[15489] = {X 83.3127, Y 48.2614, Z -3.0000, A 0.000, B 0.000, C 0.000 }
gfCNCPoint2[15490] = {X 82.6547, Y 47.6088, Z -3.0000, A 0.000, B 0.000, C 0.000 }
gfCNCPoint2[15491] = {X 82.1576, Y 46.8267, Z -3.0000, A 0.000, B 0.000, C 0.000 }
gfCNCPoint2[15492] = {X 81.8459, Y 45.9539, Z -3.0000, A 0.000, B 0.000, C 0.000 }
gfCNCPoint2[15493] = {X 81.7352, Y 45.0338, Z -3.0000, A 0.000, B 0.000, C 0.000 }
gfCNCPoint2[15494] = {X 81.7351, Y 44.2079, Z -3.0000, A 0.000, B 0.000, C 0.000 }
gfCNCPoint2[15495] = {X 81.8409, Y 43.2949, Z -3.0000, A 0.000, B 0.000, C 0.000 }
gfCNCPoint2[15496] = {X 82.1418, Y 42.4264, Z -3.0000, A 0.000, B 0.000, C 0.000 }
gfCNCPoint2[15497] = {X 82.6236, Y 41.6436, Z -3.0000, A 0.000, B 0.000, C 0.000 }
gfCNCPoint2[15498] = {X 83.2634, Y 40.9837, Z -3.0000, A 0.000, B 0.000, C 0.000 }
gfCNCPoint2[15499] = {X 83.2633, Y 28.5920, Z -3.0000, A 0.000, B 0.000, C 0.000 }
gfCNCPoint2[15500] = {X 79.2633, Y 28.5920, Z -3.0000, A 0.000, B 0.000, C 0.000 }
gfCNCPoint2[15501] = {X 83.3433, Y 28.5920, Z -3.0000, A 0.000, B 0.000, C 0.000 }
gfCNCPoint2[15502] = {X 83.3431, Y 16.1614, Z -3.0000, A 0.000, B 0.000, C 0.000 }
gfCNCPoint2[15503] = {X 82.7058, Y 15.5226, Z -3.0000, A 0.000, B 0.000, C 0.000 }
gfCNCPoint2[15504] = {X 82.2244, Y 14.7592, Z -3.0000, A 0.000, B 0.000, C 0.000 }
gfCNCPoint2[15505] = {X 81.9227, Y 13.9088, Z -3.0000, A 0.000, B 0.000, C 0.000 }
gfCNCPoint2[15506] = {X 81.8152, Y 13.0128, Z -3.0000, A 0.000, B 0.000, C 0.000 }
gfCNCPoint2[15507] = {X 81.8151, Y 12.1868, Z -3.0000, A 0.000, B 0.000, C 0.000 }
gfCNCPoint2[15508] = {X 81.9174, Y 11.2789, Z -3.0000, A 0.000, B 0.000, C 0.000 }
gfCNCPoint2[15509] = {X 82.2191, Y 10.4166, Z -3.0000, A 0.000, B 0.000, C 0.000 }
gfCNCPoint2[15510] = {X 82.7052, Y 9.6430, Z -3.0000, A 0.000, B 0.000, C 0.000 }
gfCNCPoint2[15511] = {X 83.3512, Y 8.9969, Z -3.0000, A 0.000, B 0.000, C 0.000 }
gfCNCPoint2[15512] = {X 84.1248, Y 8.5109, Z -3.0000, A 0.000, B 0.000, C 0.000 }
gfCNCPoint2[15513] = {X 84.9872, Y 8.2091, Z -3.0000, A 0.000, B 0.000, C 0.000 }
gfCNCPoint2[15514] = {X 85.8951, Y 8.1068, Z -3.0000, A 0.000, B 0.000, C 0.000 }
gfCNCPoint2[15515] = {X 94.0497, Y 8.1068, Z -3.0000, A 0.000, B 0.000, C 0.000 }
gfCNCPoint2[15516] = {X 94.9576, Y 8.2091, Z -3.0000, A 0.000, B 0.000, C 0.000 }
gfCNCPoint2[15517] = {X 95.8199, Y 8.5109, Z -3.0000, A 0.000, B 0.000, C 0.000 }
gfCNCPoint2[15518] = {X 96.5935, Y 8.9969, Z -3.0000, A 0.000, B 0.000, C 0.000 }
gfCNCPoint2[15519] = {X 97.2395, Y 9.6430, Z -3.0000, A 0.000, B 0.000, C 0.000 }
gfCNCPoint2[15520] = {X 97.7256, Y 10.4166, Z -3.0000, A 0.000, B 0.000, C 0.000 }
gfCNCPoint2[15521] = {X 98.0274, Y 11.2789, Z -3.0000, A 0.000, B 0.000, C 0.000 }
gfCNCPoint2[15522] = {X 98.1297, Y 12.1868, Z -3.0000, A 0.000, B 0.000, C 0.000 }
gfCNCPoint2[15523] = {X 98.1297, Y 12.9781, Z -3.0000, A 0.000, B 0.000, C 0.000 }
gfCNCPoint2[15524] = {X 98.0631, Y 13.7122, Z -3.0000, A 0.000, B 0.000, C 0.000 }
gfCNCPoint2[15525] = {X 97.8655, Y 14.4223, Z -3.0000, A 0.000, B 0.000, C 0.000 }
gfCNCPoint2[15526] = {X 97.5434, Y 15.0853, Z -3.0000, A 0.000, B 0.000, C 0.000 }
gfCNCPoint2[15527] = {X 97.4970, Y 15.1603, Z -3.0000, A 0.000, B 0.000, C 0.000 }
gfCNCPoint2[15528] = {X 97.4491, Y 15.2342, Z -3.0000, A 0.000, B 0.000, C 0.000 }
gfCNCPoint2[15529] = {X 97.4847, Y 15.2810, Z -3.0000, A 0.000, B 0.000, C 0.000 }
gfCNCPoint2[15530] = {X 101.8768, Y 26.1688, Z -3.0000, A 0.000, B 0.000, C 0.000 }
gfCNCPoint2[15531] = {X 102.0527, Y 25.7389, Z -3.0000, A 0.000, B 0.000, C 0.000 }
gfCNCPoint2[15532] = {X 106.2850, Y 15.1978, Z -3.0000, A 0.000, B 0.000, C 0.000 }
gfCNCPoint2[15533] = {X 106.2416, Y 15.1294, Z -3.0000, A 0.000, B 0.000, C 0.000 }
gfCNCPoint2[15534] = {X 106.1996, Y 15.0602, Z -3.0000, A 0.000, B 0.000, C 0.000 }
gfCNCPoint2[15535] = {X 105.8900, Y 14.4158, Z -3.0000, A 0.000, B 0.000, C 0.000 }
gfCNCPoint2[15536] = {X 105.6977, Y 13.7272, Z -3.0000, A 0.000, B 0.000, C 0.000 }
gfCNCPoint2[15537] = {X 105.6285, Y 13.0157, Z -3.0000, A 0.000, B 0.000, C 0.000 }
gfCNCPoint2[15538] = {X 105.6283, Y 12.1868, Z -3.0000, A 0.000, B 0.000, C 0.000 }
gfCNCPoint2[15539] = {X 105.7306, Y 11.2789, Z -3.0000, A 0.000, B 0.000, C 0.000 }
gfCNCPoint2[15540] = {X 106.0323, Y 10.4166, Z -3.0000, A 0.000, B 0.000, C 0.000 }
gfCNCPoint2[15541] = {X 106.5184, Y 9.6430, Z -3.0000, A 0.000, B 0.000, C 0.000 }
gfCNCPoint2[15542] = {X 107.1644, Y 8.9969, Z -3.0000, A 0.000, B 0.000, C 0.000 }
gfCNCPoint2[15543] = {X 107.9380, Y 8.5109, Z -3.0000, A 0.000, B 0.000, C 0.000 }
gfCNCPoint2[15544] = {X 108.8004, Y 8.2091, Z -3.0000, A 0.000, B 0.000, C 0.000 }
gfCNCPoint2[15545] = {X 109.7083, Y 8.1068, Z -3.0000, A 0.000, B 0.000, C 0.000 }
gfCNCPoint2[15546] = {X 117.7916, Y 8.1068, Z -3.0000, A 0.000, B 0.000, C 0.000 }
gfCNCPoint2[15547] = {X 118.6995, Y 8.2091, Z -3.0000, A 0.000, B 0.000, C 0.000 }
gfCNCPoint2[15548] = {X 119.5618, Y 8.5109, Z -3.0000, A 0.000, B 0.000, C 0.000 }
gfCNCPoint2[15549] = {X 120.3354, Y 8.9969, Z -3.0000, A 0.000, B 0.000, C 0.000 }
gfCNCPoint2[15550] = {X 120.9814, Y 9.6430, Z -3.0000, A 0.000, B 0.000, C 0.000 }
gfCNCPoint2[15551] = {X 121.4675, Y 10.4166, Z -3.0000, A 0.000, B 0.000, C 0.000 }
gfCNCPoint2[15552] = {X 121.7693, Y 11.2789, Z -3.0000, A 0.000, B 0.000, C 0.000 }
gfCNCPoint2[15553] = {X 121.8716, Y 12.1868, Z -3.0000, A 0.000, B 0.000, C 0.000 }
gfCNCPoint2[15554] = {X 121.8716, Y 12.9781, Z -3.0000, A 0.000, B 0.000, C 0.000 }
gfCNCPoint2[15555] = {X 121.7699, Y 13.8831, Z -3.0000, A 0.000, B 0.000, C 0.000 }
gfCNCPoint2[15556] = {X 121.4701, Y 14.7430, Z -3.0000, A 0.000, B 0.000, C 0.000 }
gfCNCPoint2[15557] = {X 120.9870, Y 15.5149, Z -3.0000, A 0.000, B 0.000, C 0.000 }
gfCNCPoint2[15558] = {X 120.3447, Y 16.1605, Z -3.0000, A 0.000, B 0.000, C 0.000 }
gfCNCPoint2[15559] = {X 120.3434, Y 41.0281, Z -3.0000, A 0.000, B 0.000, C 0.000 }
gfCNCPoint2[15560] = {X 120.4675, Y 41.1289, Z -3.0000, A 0.000, B 0.000, C 0.000 }
gfCNCPoint2[15561] = {X 121.0552, Y 41.7603, Z -3.0000, A 0.000, B 0.000, C 0.000 }
gfCNCPoint2[15562] = {X 121.4970, Y 42.5012, Z -3.0000, A 0.000, B 0.000, C 0.000 }
gfCNCPoint2[15563] = {X 121.7732, Y 43.3184, Z -3.0000, A 0.000, B 0.000, C 0.000 }
gfCNCPoint2[15564] = {X 121.8714, Y 44.1754, Z -3.0000, A 0.000, B 0.000, C 0.000 }
gfCNCPoint2[15565] = {X 121.8716, Y 45.0000, Z -3.0000, A 0.000, B 0.000, C 0.000 }
gfCNCPoint2[15566] = {X 121.7693, Y 45.9079, Z -3.0000, A 0.000, B 0.000, C 0.000 }
gfCNCPoint2[15567] = {X 121.4675, Y 46.7702, Z -3.0000, A 0.000, B 0.000, C 0.000 }
gfCNCPoint2[15568] = {X 120.9814, Y 47.5438, Z -3.0000, A 0.000, B 0.000, C 0.000 }
gfCNCPoint2[15569] = {X 120.3354, Y 48.1899, Z -3.0000, A 0.000, B 0.000, C 0.000 }
gfCNCPoint2[15570] = {X 119.5618, Y 48.6760, Z -3.0000, A 0.000, B 0.000, C 0.000 }
gfCNCPoint2[15571] = {X 118.6995, Y 48.9777, Z -3.0000, A 0.000, B 0.000, C 0.000 }
gfCNCPoint2[15572] = {X 117.7916, Y 49.0800, Z -3.0000, A 0.000, B 0.000, C 0.000 }
gfCNCPoint2[15573] = {X 111.9185, Y 49.0800, Z -3.0000, A 0.000, B 0.000, C 0.000 }
gfCNCPoint2[15574] = {X 111.0151, Y 48.9787, Z -3.0000, A 0.000, B 0.000, C 0.000 }
gfCNCPoint2[15575] = {X 110.1565, Y 48.6799, Z -3.0000, A 0.000, B 0.000, C 0.000 }
gfCNCPoint2[15576] = {X 109.3855, Y 48.1985, Z -3.0000, A 0.000, B 0.000, C 0.000 }
gfCNCPoint2[15577] = {X 108.7401, Y 47.5582, Z -3.0000, A 0.000, B 0.000, C 0.000 }
gfCNCPoint2[15578] = {X 108.2526, Y 46.7909, Z -3.0000, A 0.000, B 0.000, C 0.000 }
gfCNCPoint2[15579] = {X 107.9470, Y 45.9348, Z -3.0000, A 0.000, B 0.000, C 0.000 }
gfCNCPoint2[15580] = {X 107.8386, Y 45.0322, Z -3.0000, A 0.000, B 0.000, C 0.000 }
gfCNCPoint2[15581] = {X 107.8385, Y 44.1811, Z -3.0000, A 0.000, B 0.000, C 0.000 }
gfCNCPoint2[15582] = {X 107.8724, Y 43.6671, Z -3.0000, A 0.000, B 0.000, C 0.000 }
gfCNCPoint2[15583] = {X 107.9734, Y 43.1619, Z -3.0000, A 0.000, B 0.000, C 0.000 }
gfCNCPoint2[15584] = {X 108.1303, Y 42.6977, Z -3.0000, A 0.000, B 0.000, C 0.000 }
gfCNCPoint2[15585] = {X 108.3438, Y 42.2566, Z -3.0000, A 0.000, B 0.000, C 0.000 }
gfCNCPoint2[15586] = {X 108.8072, Y 41.5728, Z -3.0000, A 0.000, B 0.000, C 0.000 }
gfCNCPoint2[15587] = {X 109.3666, Y 40.9650, Z -3.0000, A 0.000, B 0.000, C 0.000 }
gfCNCPoint2[15588] = {X 109.3665, Y 39.0029, Z -3.0000, A 0.000, B 0.000, C 0.000 }
gfCNCPoint2[15589] = {X 108.9865, Y 39.0029, Z -3.0000, A 0.000, B 0.000, C 0.000 }
gfCNCPoint2[15590] = {X 105.8902, Y 46.5692, Z -3.0000, A 0.000, B 0.000, C 0.000 }
gfCNCPoint2[15591] = {X 105.5407, Y 47.2300, Z -3.0000, A 0.000, B 0.000, C 0.000 }
gfCNCPoint2[15592] = {X 105.0765, Y 47.8159, Z -3.0000, A 0.000, B 0.000, C 0.000 }
gfCNCPoint2[15593] = {X 104.5133, Y 48.3073, Z -3.0000, A 0.000, B 0.000, C 0.000 }
gfCNCPoint2[15594] = {X 103.8698, Y 48.6877, Z -3.0000, A 0.000, B 0.000, C 0.000 }
gfCNCPoint2[15595] = {X 102.9784, Y 48.9895, Z -3.0000, A 0.000, B 0.000, C 0.000 }
gfCNCPoint2[15596] = {X 102.0417, Y 49.0792, Z -3.0000, A 0.000, B 0.000, C 0.000 }
gfCNCPoint2[15597] = {X 101.1093, Y 48.9518, Z -3.0000, A 0.000, B 0.000, C 0.000 }
gfCNCPoint2[15598] = {X 100.2309, Y 48.6142, Z -3.0000, A 0.000, B 0.000, C 0.000 }
gfCNCPoint2[15599] = {X 99.4532, Y 48.0843, Z -3.0000, A 0.000, B 0.000, C 0.000 }
gfCNCPoint2[15600] = {X 98.8176, Y 47.3903, Z -3.0000, A 0.000, B 0.000, C 0.000 }
gfCNCPoint2[15601] = {X 98.3579, Y 46.5692, Z -3.0000, A 0.000, B 0.000, C 0.000 }
gfCNCPoint2[15602] = {X 94.8915, Y 38.0918, Z -3.0000, A 0.000, B 0.000, C 0.000 }
gfCNCPoint2[15603] = {X 94.8903, Y 38.2310, Z -3.0000, A 0.000, B 0.000, C 0.000 }
gfCNCPoint2[15604] = {X 94.8905, Y 41.0172, Z -3.0000, A 0.000, B 0.000, C 0.000 }
gfCNCPoint2[15605] = {X 95.4392, Y 41.5580, Z -3.0000, A 0.000, B 0.000, C 0.000 }
gfCNCPoint2[15606] = {X 95.8788, Y 42.1907, Z -3.0000, A 0.000, B 0.000, C 0.000 }
gfCNCPoint2[15607] = {X 96.1088, Y 42.6650, Z -3.0000, A 0.000, B 0.000, C 0.000 }
gfCNCPoint2[15608] = {X 96.2770, Y 43.1645, Z -3.0000, A 0.000, B 0.000, C 0.000 }
gfCNCPoint2[15609] = {X 96.3809, Y 43.6819, Z -3.0000, A 0.000, B 0.000, C 0.000 }
gfCNCPoint2[15610] = {X 96.4185, Y 44.2083, Z -3.0000, A 0.000, B 0.000, C 0.000 }
gfCNCPoint2[15611] = {X 96.4184, Y 45.0392, Z -3.0000, A 0.000, B 0.000, C 0.000 }
gfCNCPoint2[15612] = {X 96.3086, Y 45.9406, Z -3.0000, A 0.000, B 0.000, C 0.000 }
gfCNCPoint2[15613] = {X 96.0023, Y 46.7954, Z -3.0000, A 0.000, B 0.000, C 0.000 }
gfCNCPoint2[15614] = {X 95.5144, Y 47.5613, Z -3.0000, A 0.000, B 0.000, C 0.000 }
gfCNCPoint2[15615] = {X 94.8692, Y 48.2003, Z -3.0000, A 0.000, B 0.000, C 0.000 }
gfCNCPoint2[15616] = {X 94.0987, Y 48.6808, Z -3.0000, A 0.000, B 0.000, C 0.000 }
gfCNCPoint2[15617] = {X 93.2410, Y 48.9789, Z -3.0000, A 0.000, B 0.000, C 0.000 }
gfCNCPoint2[15618] = {X 92.3385, Y 49.0800, Z -3.0000, A 0.000, B 0.000, C 0.000 }
gfCNCPoint2[15619] = {X 85.8951, Y 49.0800, Z -3.0000, A 0.000, B 0.000, C 0.000 }
gfCNCPoint2[15620] = {X 84.9918, Y 48.9788, Z -3.0000, A 0.000, B 0.000, C 0.000 }
gfCNCPoint2[15621] = {X 84.1334, Y 48.6801, Z -3.0000, A 0.000, B 0.000, C 0.000 }
gfCNCPoint2[15622] = {X 83.3624, Y 48.1987, Z -3.0000, A 0.000, B 0.000, C 0.000 }
gfCNCPoint2[15623] = {X 82.7171, Y 47.5586, Z -3.0000, A 0.000, B 0.000, C 0.000 }
gfCNCPoint2[15624] = {X 82.2295, Y 46.7916, Z -3.0000, A 0.000, B 0.000, C 0.000 }
gfCNCPoint2[15625] = {X 81.9238, Y 45.9356, Z -3.0000, A 0.000, B 0.000, C 0.000 }
gfCNCPoint2[15626] = {X 81.8152, Y 45.0332, Z -3.0000, A 0.000, B 0.000, C 0.000 }
gfCNCPoint2[15627] = {X 81.8151, Y 44.2084, Z -3.0000, A 0.000, B 0.000, C 0.000 }
gfCNCPoint2[15628] = {X 81.9210, Y 43.3035, Z -3.0000, A 0.000, B 0.000, C 0.000 }
gfCNCPoint2[15629] = {X 82.2222, Y 42.4437, Z -3.0000, A 0.000, B 0.000, C 0.000 }
gfCNCPoint2[15630] = {X 82.7041, Y 41.6706, Z -3.0000, A 0.000, B 0.000, C 0.000 }
gfCNCPoint2[15631] = {X 83.3434, Y 41.0216, Z -3.0000, A 0.000, B 0.000, C 0.000 }
gfCNCPoint2[15632] = {X 83.3433, Y 28.5920, Z -3.0000, A 0.000, B 0.000, C 0.000 }
gfCNCPoint2[15633] = {X 79.3433, Y 28.5920, Z -3.0000, A 0.000, B 0.000, C 0.000 }
gfCNCPoint2[15634] = {X 83.4233, Y 28.5920, Z -3.0000, A 0.000, B 0.000, C 0.000 }
gfCNCPoint2[15635] = {X 83.4231, Y 16.1228, Z -3.0000, A 0.000, B 0.000, C 0.000 }
gfCNCPoint2[15636] = {X 82.7809, Y 15.4884, Z -3.0000, A 0.000, B 0.000, C 0.000 }
gfCNCPoint2[15637] = {X 82.2973, Y 14.7261, Z -3.0000, A 0.000, B 0.000, C 0.000 }
gfCNCPoint2[15638] = {X 81.9969, Y 13.8749, Z -3.0000, A 0.000, B 0.000, C 0.000 }
gfCNCPoint2[15639] = {X 81.8951, Y 12.9779, Z -3.0000, A 0.000, B 0.000, C 0.000 }
gfCNCPoint2[15640] = {X 81.8951, Y 12.1868, Z -3.0000, A 0.000, B 0.000, C 0.000 }
gfCNCPoint2[15641] = {X 81.9954, Y 11.2967, Z -3.0000, A 0.000, B 0.000, C 0.000 }
gfCNCPoint2[15642] = {X 82.2912, Y 10.4513, Z -3.0000, A 0.000, B 0.000, C 0.000 }
gfCNCPoint2[15643] = {X 82.7677, Y 9.6929, Z -3.0000, A 0.000, B 0.000, C 0.000 }
gfCNCPoint2[15644] = {X 83.4011, Y 9.0595, Z -3.0000, A 0.000, B 0.000, C 0.000 }
gfCNCPoint2[15645] = {X 84.1595, Y 8.5829, Z -3.0000, A 0.000, B 0.000, C 0.000 }
gfCNCPoint2[15646] = {X 85.0050, Y 8.2871, Z -3.0000, A 0.000, B 0.000, C 0.000 }
gfCNCPoint2[15647] = {X 85.8951, Y 8.1868, Z -3.0000, A 0.000, B 0.000, C 0.000 }
gfCNCPoint2[15648] = {X 94.0497, Y 8.1868, Z -3.0000, A 0.000, B 0.000, C 0.000 }
